KUKA KRL program: MyProgram_075().src

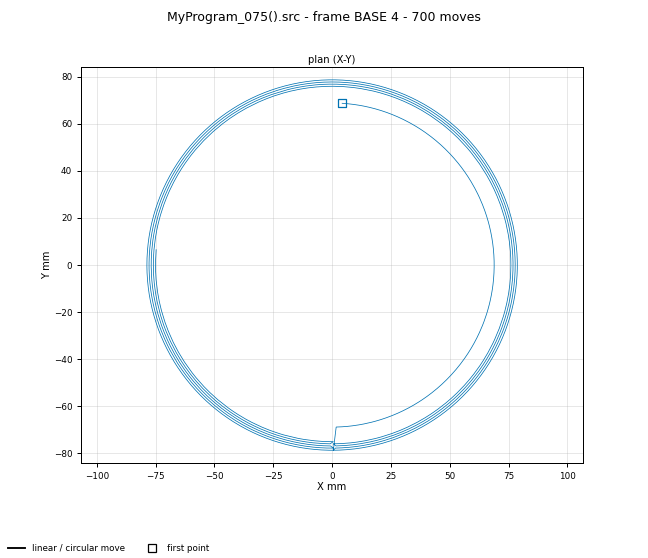
[picture p0: tool path of MyProgram_075().src in frame BASE 4, 700 of 700 moves have a stored position in this frame; points joined in program order, loops and branches not executed]
&ACCESS RVP
&REL 1
&PARAM TEMPLATE = C:\KRC\Roboter\Template\vorgabe
&PARAM EDITMASK = *
DEF MyProgram_075()
; ---- Setting reference (Base) ----
$BASE = BASE_DATA[4]

; --------------------------
; ---- Setting tool (TCP) ----
$TOOL = TOOL_DATA[3]
; --------------------------

$VEL.CP = VEL_APROX_PRINT
Startdeposition()
$VEL.CP = VEL_PRINT
LIN {X 4.2786,Y 68.757,Z 78,A 79.6597,B 24.8748,C -2.582,E1 25.012,E2 4.5437} C_DIS
LIN {X 6.8006,Y 68.5536,Z 78,A 77.5534,B 24.8748,C -2.5817,E1 25.0178,E2 6.6494} C_DIS
LIN {X 9.2868,Y 68.2614,Z 78,A 75.7343,B 24.8743,C -2.5876,E1 25.0228,E2 8.4531} C_DIS
LIN {X 11.7416,Y 67.8821,Z 78,A 73.6949,B 24.8743,C -2.5876,E1 25.0284,E2 10.4905} C_DIS
LIN {X 13.4915,Y 67.556,Z 78,A 72.2248,B 24.8743,C -2.5873,E1 25.0325,E2 11.9597} C_DIS
LIN {X 15.8736,Y 67.0363,Z 78,A 70.0908,B 24.8747,C -2.5836,E1 25.0383,E2 14.0995} C_DIS
LIN {X 18.4538,Y 66.3722,Z 78,A 67.9692,B 24.8746,C -2.5846,E1 25.044,E2 16.2154} C_DIS
LIN {X 20.828,Y 65.6662,Z 78,A 65.6223,B 24.8754,C -2.576,E1 25.0503,E2 18.5786} C_DIS
LIN {X 23.2331,Y 64.8543,Z 78,A 63.7895,B 24.8749,C -2.581,E1 25.0551,E2 20.3957} C_DIS
LIN {X 25.5953,Y 63.9589,Z 78,A 61.4087,B 24.8758,C -2.5721,E1 25.0614,E2 22.7926} C_DIS
LIN {X 27.9246,Y 62.9769,Z 78,A 59.3241,B 24.876,C -2.5702,E1 25.0667,E2 24.8765} C_DIS
LIN {X 30.2585,Y 61.8891,Z 78,A 57.1963,B 24.8762,C -2.568,E1 25.072,E2 27.0039} C_DIS
LIN {X 32.8695,Y 60.5417,Z 78,A 54.8407,B 24.8762,C -2.5671,E1 25.0779,E2 29.3552} C_DIS
LIN {X 35.4913,Y 59.0439,Z 78,A 52.275,B 24.8768,C -2.5621,E1 25.084,E2 31.9249} C_DIS
LIN {X 37.5793,Y 57.7379,Z 78,A 50.1926,B 24.8772,C -2.558,E1 25.0889,E2 34.0101} C_DIS
LIN {X 39.6743,Y 56.3189,Z 78,A 48.0936,B 24.8775,C -2.5547,E1 25.0938,E2 36.1097} C_DIS
LIN {X 42.0686,Y 54.5521,Z 78,A 45.8309,B 24.8774,C -2.5559,E1 25.0988,E2 38.3615} C_DIS
LIN {X 44.0446,Y 52.9696,Z 78,A 43.7356,B 24.8777,C -2.5522,E1 25.1033,E2 40.4575} C_DIS
LIN {X 46.2398,Y 51.0659,Z 78,A 41.2144,B 24.8784,C -2.5448,E1 25.1086,E2 42.9863} C_DIS
LIN {X 48.1387,Y 49.28,Z 78,A 38.9784,B 24.879,C -2.5386,E1 25.1131,E2 45.2277} C_DIS
LIN {X 50.2041,Y 47.1725,Z 78,A 36.7249,B 24.879,C -2.5386,E1 25.1175,E2 47.4716} C_DIS
LIN {X 51.888,Y 45.3137,Z 78,A 34.6568,B 24.8794,C -2.5344,E1 25.1213,E2 49.5403} C_DIS
LIN {X 53.5179,Y 43.3766,Z 78,A 32.5614,B 24.8799,C -2.5298,E1 25.125,E2 51.637} C_DIS
LIN {X 54.8494,Y 41.682,Z 78,A 30.5831,B 24.8807,C -2.5206,E1 25.1284,E2 53.6276} C_DIS
LIN {X 56.3431,Y 39.6397,Z 78,A 28.4879,B 24.8812,C -2.5156,E1 25.1318,E2 55.7244} C_DIS
LIN {X 57.7579,Y 37.5483,Z 78,A 26.6761,B 24.881,C -2.518,E1 25.1346,E2 57.5216} C_DIS
LIN {X 59.0958,Y 35.4055,Z 78,A 24.3033,B 24.8822,C -2.5053,E1 25.1381,E2 59.9124} C_DIS
LIN {X 60.625,Y 32.7158,Z 78,A 21.9754,B 24.8822,C -2.505,E1 25.1412,E2 62.2288} C_DIS
LIN {X 61.8865,Y 30.2638,Z 78,A 19.7787,B 24.8826,C -2.5013,E1 25.144,E2 64.4226} C_DIS
LIN {X 62.6469,Y 28.657,Z 78,A 18.0045,B 24.8837,C -2.4892,E1 25.1461,E2 66.2158} C_DIS
LIN {X 63.9379,Y 25.6469,Z 78,A 15.3278,B 24.8843,C -2.4827,E1 25.149,E2 68.8931} C_DIS
LIN {X 64.8826,Y 23.1535,Z 78,A 13.1121,B 24.8849,C -2.4763,E1 25.1511,E2 71.1115} C_DIS
LIN {X 65.6891,Y 20.7553,Z 78,A 11.0195,B 24.8855,C -2.4704,E1 25.1529,E2 73.2062} C_DIS
LIN {X 66.3949,Y 18.3737,Z 78,A 9.2251,B 24.8853,C -2.4716,E1 25.1543,E2 74.9876} C_DIS
LIN {X 66.836,Y 16.6972,Z 78,A 7.5223,B 24.8864,C -2.4601,E1 25.1555,E2 76.7076} C_DIS
LIN {X 67.3994,Y 14.2542,Z 78,A 5.7231,B 24.8863,C -2.4615,E1 25.1565,E2 78.493} C_DIS
LIN {X 67.869,Y 11.8169,Z 78,A 3.6106,B 24.887,C -2.4539,E1 25.1576,E2 80.6113} C_DIS
LIN {X 68.2635,Y 9.2719,Z 78,A 1.5451,B 24.8874,C -2.4493,E1 25.1585,E2 82.6754} C_DIS
LIN {X 68.5556,Y 6.7813,Z 78,A -0.5387,B 24.888,C -2.4428,E1 25.1591,E2 84.7622} C_DIS
LIN {X 68.7582,Y 4.2609,Z 78,A -2.6227,B 24.8886,C -2.4367,E1 25.1595,E2 86.8483} C_DIS
LIN {X 68.8683,Y 1.734,Z 78,A -4.7221,B 24.8892,C -2.4302,E1 25.1598,E2 88.9506} C_DIS
LIN {X 68.8856,Y -0.7727,Z 78,A -6.777,B 24.8897,C -2.4244,E1 25.1598,E2 91.007} C_DIS
LIN {X 68.8078,Y -3.3703,Z 78,A -8.9237,B 24.8903,C -2.4179,E1 25.1595,E2 93.1562} C_DIS
LIN {X 68.6402,Y -5.8623,Z 78,A -10.9954,B 24.8909,C -2.4114,E1 25.1591,E2 95.2308} C_DIS
LIN {X 68.3768,Y -8.3944,Z 78,A -13.0575,B 24.8913,C -2.4062,E1 25.1585,E2 97.2931} C_DIS
LIN {X 68.1372,Y -10.1567,Z 78,A -14.8223,B 24.8925,C -2.3937,E1 25.1578,E2 99.077} C_DIS
LIN {X 67.7274,Y -12.6047,Z 78,A -16.5998,B 24.8924,C -2.395,E1 25.1569,E2 100.841} C_DIS
LIN {X 67.2192,Y -15.0813,Z 78,A -18.6632,B 24.8929,C -2.3895,E1 25.1557,E2 102.9055} C_DIS
LIN {X 66.8248,Y -16.7427,Z 78,A -20.1027,B 24.8933,C -2.3845,E1 25.1548,E2 104.3485} C_DIS
LIN {X 66.1771,Y -19.1423,Z 78,A -22.1623,B 24.8939,C -2.3783,E1 25.1532,E2 106.411} C_DIS
LIN {X 65.6458,Y -20.8911,Z 78,A -23.9282,B 24.8949,C -2.3668,E1 25.1517,E2 108.1938} C_DIS
LIN {X 64.5825,Y -23.9782,Z 78,A -26.3411,B 24.8949,C -2.3668,E1 25.1495,E2 110.5934} C_DIS
LIN {X 63.9437,Y -25.6327,Z 78,A -28.0923,B 24.896,C -2.3548,E1 25.1477,E2 112.3632} C_DIS
LIN {X 62.6548,Y -28.6393,Z 78,A -30.5251,B 24.896,C -2.3545,E1 25.145,E2 114.7834} C_DIS
LIN {X 61.5438,Y -30.9551,Z 78,A -32.8114,B 24.8969,C -2.3441,E1 25.1421,E2 117.082} C_DIS
LIN {X 60.331,Y -33.2567,Z 78,A -34.7671,B 24.8969,C -2.3434,E1 25.1396,E2 119.029} C_DIS
LIN {X 59.111,Y -35.3799,Z 78,A -37.0001,B 24.8979,C -2.3323,E1 25.1364,E2 121.2768} C_DIS
LIN {X 57.7275,Y -37.5951,Z 78,A -39.257,B 24.8987,C -2.3239,E1 25.133,E2 123.5421} C_DIS
LIN {X 56.3166,Y -39.6775,Z 78,A -41.3446,B 24.8992,C -2.3183,E1 25.1297,E2 125.6327} C_DIS
LIN {X 54.5098,Y -42.1235,Z 78,A -43.8424,B 24.8997,C -2.3124,E1 25.1255,E2 128.1325} C_DIS
LIN {X 52.7111,Y -44.3556,Z 78,A -46.1758,B 24.9001,C -2.3076,E1 25.1213,E2 130.4666} C_DIS
LIN {X 50.7147,Y -46.6232,Z 78,A -48.7308,B 24.9007,C -2.3002,E1 25.1165,E2 133.0277} C_DIS
LIN {X 48.6926,Y -48.7328,Z 78,A -51.1426,B 24.9012,C -2.2948,E1 25.1118,E2 135.4421} C_DIS
LIN {X 46.5721,Y -50.7616,Z 78,A -53.3854,B 24.9012,C -2.2944,E1 25.1072,E2 137.6766} C_DIS
LIN {X 44.6488,Y -52.4613,Z 78,A -55.7017,B 24.9021,C -2.2847,E1 25.1023,E2 140.0066} C_DIS
LIN {X 42.3702,Y -54.3197,Z 78,A -57.8465,B 24.9018,C -2.2874,E1 25.0977,E2 142.1372} C_DIS
LIN {X 40.358,Y -55.831,Z 78,A -59.9287,B 24.9022,C -2.2833,E1 25.093,E2 144.2215} C_DIS
LIN {X 38.2711,Y -57.2817,Z 78,A -62.0044,B 24.9025,C -2.2801,E1 25.0882,E2 146.2977} C_DIS
LIN {X 36.8169,Y -58.2268,Z 78,A -63.7389,B 24.9034,C -2.2698,E1 25.0841,E2 148.0511} C_DIS
LIN {X 34.6799,Y -59.5246,Z 78,A -65.547,B 24.9031,C -2.273,E1 25.0798,E2 149.8459} C_DIS
LIN {X 32.4785,Y -60.7538,Z 78,A -67.8751,B 24.9039,C -2.2634,E1 25.0741,E2 152.1901} C_DIS
LIN {X 30.1975,Y -61.9191,Z 78,A -70.0366,B 24.9043,C -2.2592,E1 25.0686,E2 154.3557} C_DIS
LIN {X 27.9116,Y -62.9827,Z 78,A -71.8452,B 24.9039,C -2.2634,E1 25.0641,E2 156.1498} C_DIS
LIN {X 25.5875,Y -63.9621,Z 78,A -74.2251,B 24.9048,C -2.2532,E1 25.0579,E2 158.5485} C_DIS
LIN {X 23.1567,Y -64.8814,Z 78,A -76.352,B 24.9049,C -2.2512,E1 25.0523,E2 160.6755} C_DIS
LIN {X 20.757,Y -65.6885,Z 78,A -78.4536,B 24.9051,C -2.2488,E1 25.0467,E2 162.7789} C_DIS
LIN {X 18.3446,Y -66.4028,Z 78,A -80.2786,B 24.9047,C -2.2533,E1 25.0419,E2 164.5902} C_DIS
LIN {X 16.6718,Y -66.8422,Z 78,A -81.9846,B 24.9054,C -2.2451,E1 25.0372,E2 166.313} C_DIS
LIN {X 13.475,Y -67.5594,Z 78,A -84.4101,B 24.905,C -2.2502,E1 25.0306,E2 168.7233} C_DIS
LIN {X 11.3377,Y -67.9497,Z 78,A -86.3388,B 24.9054,C -2.2458,E1 25.0253,E2 170.6604} C_DIS
LIN {X 8.4843,Y -68.3656,Z 78,A -88.6117,B 24.9053,C -2.2473,E1 25.019,E2 172.9278} C_DIS
LIN {X 6.699,Y -68.5635,Z 78,A -90.3546,B 24.9058,C -2.2403,E1 25.0141,E2 174.6862} C_DIS
LIN {X 4.2094,Y -68.7615,Z 78,A -92.2011,B 24.9054,C -2.245,E1 25.009,E2 176.5206} C_DIS
LIN {X 1.7291,Y -68.8684,Z 78,A -94.2379,B 24.9054,C -2.245,E1 25.0033,E2 178.557} C_DIS
LIN {X 1.7291,Y -68.8684,Z 78,A -94.2379,B 24.9054,C -2.245,E1 25.0033,E2 178.557} C_DIS
Enddeposition()
LIN {X 0.524,Y -78.7317,Z 79,A -94.3644,B 24.917,C -2.1042,E1 25.002,E2 179.0178} C_DIS
Startdeposition()
$VEL.CP = VEL_PRINT
LIN {X -1.339,Y -78.7246,Z 79,A -96.4259,B 24.9186,C -2.0837,E1 24.9962,E2 181.1278} C_DIS
LIN {X -4.456,Y -78.6098,Z 79,A -98.6122,B 24.9184,C -2.0859,E1 24.9901,E2 183.3094} C_DIS
LIN {X -7.2304,Y -78.4032,Z 79,A -100.6782,B 24.9184,C -2.0848,E1 24.9843,E2 185.379} C_DIS
LIN {X -10.008,Y -78.0973,Z 79,A -102.7545,B 24.9186,C -2.0839,E1 24.9785,E2 187.4588} C_DIS
LIN {X -13.0934,Y -77.6397,Z 79,A -105.1259,B 24.9187,C -2.0817,E1 24.972,E2 189.8376} C_DIS
LIN {X -16.3074,Y -77.0302,Z 79,A -107.5052,B 24.9187,C -2.0826,E1 24.9655,E2 192.2173} C_DIS
LIN {X -19.4927,Y -76.2849,Z 79,A -109.7919,B 24.9184,C -2.0865,E1 24.9593,E2 194.498} C_DIS
LIN {X -22.4988,Y -75.453,Z 79,A -111.9817,B 24.9181,C -2.0902,E1 24.9534,E2 196.6825} C_DIS
LIN {X -25.2608,Y -74.5738,Z 79,A -114.0947,B 24.9179,C -2.0917,E1 24.9478,E2 198.7958} C_DIS
LIN {X -27.9886,Y -73.5935,Z 79,A -116.3922,B 24.9182,C -2.0885,E1 24.9418,E2 201.1057} C_DIS
LIN {X -31.0219,Y -72.3686,Z 79,A -118.7414,B 24.9179,C -2.0917,E1 24.9357,E2 203.4526} C_DIS
LIN {X -33.6646,Y -71.1778,Z 79,A -120.8891,B 24.9179,C -2.093,E1 24.9303,E2 205.6024} C_DIS
LIN {X -36.2616,Y -69.8904,Z 79,A -123.0044,B 24.9177,C -2.0955,E1 24.925,E2 207.7175} C_DIS
LIN {X -39.1328,Y -68.3226,Z 79,A -125.2953,B 24.9172,C -2.1011,E1 24.9194,E2 210.0017} C_DIS
LIN {X -41.8081,Y -66.7191,Z 79,A -127.4889,B 24.9168,C -2.1065,E1 24.9142,E2 212.1894} C_DIS
LIN {X -44.2355,Y -65.135,Z 79,A -129.7901,B 24.9169,C -2.1047,E1 24.9088,E2 214.5023} C_DIS
LIN {X -46.9038,Y -63.2425,Z 79,A -132.1761,B 24.9166,C -2.1086,E1 24.9034,E2 216.8875} C_DIS
LIN {X -49.1998,Y -61.4732,Z 79,A -134.2939,B 24.9163,C -2.1121,E1 24.8988,E2 219.0047} C_DIS
LIN {X -51.4291,Y -59.6206,Z 79,A -136.4121,B 24.916,C -2.1159,E1 24.8943,E2 221.1222} C_DIS
LIN {X -53.5887,Y -57.6873,Z 79,A -138.5308,B 24.9157,C -2.1198,E1 24.8899,E2 223.2401} C_DIS
LIN {X -55.9377,Y -55.4105,Z 79,A -140.8254,B 24.9152,C -2.127,E1 24.8854,E2 225.5272} C_DIS
LIN {X -58.0885,Y -53.1515,Z 79,A -143.0217,B 24.9146,C -2.1338,E1 24.8812,E2 227.7169} C_DIS
LIN {X -60.0055,Y -50.9774,Z 79,A -145.3272,B 24.9146,C -2.1335,E1 24.877,E2 230.0334} C_DIS
LIN {X -61.9167,Y -48.6387,Z 79,A -147.5039,B 24.9142,C -2.1392,E1 24.8732,E2 232.2067} C_DIS
LIN {X -63.8133,Y -46.1242,Z 79,A -149.8376,B 24.9138,C -2.1437,E1 24.8693,E2 234.5411} C_DIS
LIN {X -65.673,Y -43.4329,Z 79,A -152.1344,B 24.9132,C -2.1518,E1 24.8657,E2 236.8298} C_DIS
LIN {X -67.2271,Y -40.9862,Z 79,A -154.2559,B 24.9127,C -2.1569,E1 24.8626,E2 238.95} C_DIS
LIN {X -68.7977,Y -38.2914,Z 79,A -156.6403,B 24.9125,C -2.1601,E1 24.8593,E2 241.3393} C_DIS
LIN {X -70.3301,Y -35.4012,Z 79,A -158.9641,B 24.9118,C -2.168,E1 24.8563,E2 243.6568} C_DIS
LIN {X -71.5855,Y -32.7886,Z 79,A -161.1545,B 24.9115,C -2.1718,E1 24.8537,E2 245.8499} C_DIS
LIN {X -72.7439,Y -30.1315,Z 79,A -163.2772,B 24.9111,C -2.1775,E1 24.8514,E2 247.9708} C_DIS
LIN {X -73.8036,Y -27.4336,Z 79,A -165.4003,B 24.9106,C -2.1832,E1 24.8493,E2 250.0921} C_DIS
LIN {X -74.7634,Y -24.6985,Z 79,A -167.5235,B 24.9101,C -2.1891,E1 24.8474,E2 252.2134} C_DIS
LIN {X -75.7234,Y -21.5712,Z 79,A -169.8226,B 24.9094,C -2.1982,E1 24.8456,E2 254.5039} C_DIS
LIN {X -76.5184,Y -18.5551,Z 79,A -172.209,B 24.909,C -2.2022,E1 24.8439,E2 256.8948} C_DIS
LIN {X -77.2245,Y -15.3609,Z 79,A -174.6022,B 24.9085,C -2.2092,E1 24.8426,E2 259.2855} C_DIS
LIN {X -77.7375,Y -12.5081,Z 79,A -176.7265,B 24.9079,C -2.2154,E1 24.8416,E2 261.4077} C_DIS
LIN {X -78.1452,Y -9.6383,Z 79,A -178.8507,B 24.9074,C -2.2216,E1 24.8408,E2 263.5297} C_DIS
LIN {X -78.4768,Y -6.3838,Z 79,A 178.8495,B 24.9066,C -2.2311,E1 24.8402,E2 265.8206} C_DIS
LIN {X -78.668,Y -3.2706,Z 79,A 176.6473,B 24.9059,C -2.2399,E1 24.8399,E2 268.015} C_DIS
LIN {X -78.7351,Y -0.3728,Z 79,A 174.3378,B 24.9057,C -2.2417,E1 24.8398,E2 270.3341} C_DIS
LIN {X -78.684,Y 2.8981,Z 79,A 171.944,B 24.9051,C -2.2489,E1 24.84,E2 272.7252} C_DIS
LIN {X -78.4943,Y 6.1639,Z 79,A 169.6436,B 24.9043,C -2.2585,E1 24.8404,E2 275.0165} C_DIS
LIN {X -78.1886,Y 9.268,Z 79,A 167.4412,B 24.9036,C -2.2673,E1 24.841,E2 277.2109} C_DIS
LIN {X -77.8282,Y 11.9216,Z 79,A 165.395,B 24.9032,C -2.2711,E1 24.8419,E2 279.2603} C_DIS
LIN {X -77.295,Y 14.9948,Z 79,A 163.1928,B 24.9025,C -2.28,E1 24.8429,E2 281.4544} C_DIS
LIN {X -76.6907,Y 17.8297,Z 79,A 160.8836,B 24.9023,C -2.2817,E1 24.8444,E2 283.7731} C_DIS
LIN {X -75.8852,Y 21.0003,Z 79,A 158.4898,B 24.9017,C -2.2888,E1 24.8461,E2 286.1639} C_DIS
LIN {X -75.0608,Y 23.7792,Z 79,A 156.3656,B 24.9012,C -2.295,E1 24.8478,E2 288.2855} C_DIS
LIN {X -74.1347,Y 26.5258,Z 79,A 154.242,B 24.9007,C -2.3011,E1 24.8498,E2 290.4066} C_DIS
LIN {X -72.9676,Y 29.5818,Z 79,A 151.9425,B 24.8999,C -2.3103,E1 24.8521,E2 292.697} C_DIS
LIN {X -71.7539,Y 32.415,Z 79,A 149.5721,B 24.8995,C -2.3139,E1 24.8548,E2 295.0719} C_DIS
LIN {X -70.3301,Y 35.4012,Z 79,A 147.2313,B 24.8988,C -2.3226,E1 24.8576,E2 297.4045} C_DIS
LIN {X -68.9795,Y 37.9659,Z 79,A 145.1083,B 24.8983,C -2.3283,E1 24.8604,E2 299.5251} C_DIS
LIN {X -67.5353,Y 40.4791,Z 79,A 142.9176,B 24.8979,C -2.3323,E1 24.8635,E2 301.7176} C_DIS
LIN {X -65.7944,Y 43.2487,Z 79,A 140.6195,B 24.8972,C -2.341,E1 24.867,E2 304.0066} C_DIS
LIN {X -64.0298,Y 45.8207,Z 79,A 138.2347,B 24.8969,C -2.3443,E1 24.8708,E2 306.3952} C_DIS
LIN {X -62.0723,Y 48.4417,Z 79,A 135.9114,B 24.8962,C -2.352,E1 24.8747,E2 308.7112} C_DIS
LIN {X -60.2473,Y 50.6936,Z 79,A 133.722,B 24.8959,C -2.3554,E1 24.8786,E2 310.9025} C_DIS
LIN {X -58.3406,Y 52.8768,Z 79,A 131.601,B 24.8955,C -2.3604,E1 24.8826,E2 313.0211} C_DIS
LIN {X -56.0928,Y 55.2535,Z 79,A 129.3047,B 24.8947,C -2.3683,E1 24.887,E2 315.3085} C_DIS
LIN {X -53.8603,Y 57.4319,Z 79,A 127.1065,B 24.8941,C -2.3755,E1 24.8914,E2 317.4988} C_DIS
LIN {X -51.7099,Y 59.3754,Z 79,A 124.9864,B 24.8937,C -2.3799,E1 24.8958,E2 319.6166} C_DIS
LIN {X -49.6608,Y 61.0996,Z 79,A 122.9445,B 24.8935,C -2.3818,E1 24.9002,E2 321.6618} C_DIS
LIN {X -47.3783,Y 62.886,Z 79,A 120.8252,B 24.8932,C -2.386,E1 24.9049,E2 323.7789} C_DIS
LIN {X -44.8504,Y 64.7132,Z 79,A 118.4443,B 24.893,C -2.3877,E1 24.9104,E2 326.164} C_DIS
LIN {X -42.1243,Y 66.5216,Z 79,A 116.0571,B 24.8926,C -2.392,E1 24.9159,E2 328.5487} C_DIS
LIN {X -39.6473,Y 68.027,Z 79,A 113.9774,B 24.8922,C -2.3965,E1 24.9209,E2 330.6239} C_DIS
LIN {X -37.1165,Y 69.4402,Z 79,A 111.8299,B 24.892,C -2.3991,E1 24.9262,E2 332.7714} C_DIS
LIN {X -34.1995,Y 70.9207,Z 79,A 109.5301,B 24.8915,C -2.405,E1 24.9319,E2 335.0632} C_DIS
LIN {X -31.3636,Y 72.2196,Z 79,A 107.3364,B 24.891,C -2.4103,E1 24.9375,E2 337.2495} C_DIS
LIN {X -28.6842,Y 73.3251,Z 79,A 105.2206,B 24.8907,C -2.4131,E1 24.943,E2 339.3635} C_DIS
LIN {X -25.9659,Y 74.3312,Z 79,A 103.105,B 24.8905,C -2.4156,E1 24.9485,E2 341.4774} C_DIS
LIN {X -23.2123,Y 75.2366,Z 79,A 100.806,B 24.8907,C -2.413,E1 24.9547,E2 343.7866} C_DIS
LIN {X -20.0675,Y 76.1372,Z 79,A 98.4236,B 24.8905,C -2.4153,E1 24.9611,E2 346.1671} C_DIS
LIN {X -16.8872,Y 76.9037,Z 79,A 96.1349,B 24.8901,C -2.42,E1 24.9673,E2 348.4478} C_DIS
LIN {X -13.828,Y 77.5122,Z 79,A 93.9446,B 24.8897,C -2.4239,E1 24.9733,E2 350.6312} C_DIS
LIN {X -10.9656,Y 77.9686,Z 79,A 91.6483,B 24.8901,C -2.4203,E1 24.9796,E2 352.938} C_DIS
LIN {X -7.7176,Y 78.3582,Z 79,A 89.2683,B 24.89,C -2.4215,E1 24.9862,E2 355.3165} C_DIS
LIN {X -4.456,Y 78.6098,Z 79,A 86.9822,B 24.8896,C -2.4251,E1 24.9926,E2 357.5949} C_DIS
LIN {X -1.339,Y 78.7246,Z 79,A 84.7943,B 24.8894,C -2.428,E1 24.9987,E2 359.7762} C_DIS
LIN {X 1.339,Y 78.7246,Z 79,A 82.7613,B 24.8895,C -2.426,E1 25.0044,E2 361.8138} C_DIS
LIN {X 4.456,Y 78.6098,Z 79,A 80.5744,B 24.8893,C -2.4284,E1 25.0104,E2 363.9943} C_DIS
LIN {X 7.3464,Y 78.3925,Z 79,A 78.4655,B 24.8893,C -2.4283,E1 25.0163,E2 366.1024} C_DIS
LIN {X 10.008,Y 78.0973,Z 79,A 76.434,B 24.8896,C -2.4256,E1 25.022,E2 368.1387} C_DIS
LIN {X 13.0562,Y 77.6459,Z 79,A 74.0814,B 24.8899,C -2.4218,E1 25.0285,E2 370.498} C_DIS
LIN {X 16.3074,Y 77.0302,Z 79,A 71.6907,B 24.8899,C -2.4213,E1 25.035,E2 372.8871} C_DIS
LIN {X 19.4927,Y 76.2849,Z 79,A 69.4096,B 24.8899,C -2.4228,E1 25.0412,E2 375.1613} C_DIS
LIN {X 22.4988,Y 75.453,Z 79,A 67.0431,B 24.8902,C -2.4184,E1 25.0475,E2 377.5341} C_DIS
LIN {X 25.6141,Y 74.4547,Z 79,A 64.6703,B 24.8904,C -2.4167,E1 25.0538,E2 379.9065} C_DIS
LIN {X 28.3372,Y 73.4614,Z 79,A 62.6491,B 24.8904,C -2.4172,E1 25.0591,E2 381.922} C_DIS
LIN {X 31.0219,Y 72.3686,Z 79,A 60.4608,B 24.8908,C -2.4128,E1 25.0648,E2 384.1158} C_DIS
LIN {X 33.6542,Y 71.1826,Z 79,A 58.3643,B 24.891,C -2.4105,E1 25.0701,E2 386.2125} C_DIS
LIN {X 36.2616,Y 69.8904,Z 79,A 56.2534,B 24.8912,C -2.408,E1 25.0753,E2 388.3235} C_DIS
LIN {X 39.1328,Y 68.3226,Z 79,A 53.9766,B 24.8912,C -2.4077,E1 25.0809,E2 390.5942} C_DIS
LIN {X 41.8081,Y 66.7191,Z 79,A 51.7974,B 24.8912,C -2.407,E1 25.086,E2 392.7682} C_DIS
LIN {X 44.2355,Y 65.135,Z 79,A 49.6953,B 24.8916,C -2.4039,E1 25.0909,E2 394.8708} C_DIS
LIN {X 46.603,Y 63.4627,Z 79,A 47.5939,B 24.8919,C -2.4005,E1 25.0957,E2 396.9728} C_DIS
LIN {X 48.9073,Y 61.7044,Z 79,A 45.4929,B 24.8922,C -2.397,E1 25.1003,E2 399.0744} C_DIS
LIN {X 51.1453,Y 59.8624,Z 79,A 43.3923,B 24.8925,C -2.3933,E1 25.1048,E2 401.1757} C_DIS
LIN {X 53.3141,Y 57.9393,Z 79,A 41.2922,B 24.8929,C -2.3894,E1 25.1092,E2 403.2766} C_DIS
LIN {X 55.2535,Y 56.0928,Z 79,A 39.2694,B 24.8934,C -2.3832,E1 25.1133,E2 405.3057} C_DIS
LIN {X 57.4319,Y 53.8603,Z 79,A 37.0931,B 24.8936,C -2.3811,E1 25.1175,E2 407.4775} C_DIS
LIN {X 59.2303,Y 51.8761,Z 79,A 35.0713,B 24.8942,C -2.3745,E1 25.1213,E2 409.5059} C_DIS
LIN {X 61.2385,Y 49.4894,Z 79,A 32.8958,B 24.8944,C -2.3721,E1 25.1251,E2 411.6771} C_DIS
LIN {X 63.0186,Y 47.2019,Z 79,A 30.6151,B 24.8953,C -2.3618,E1 25.129,E2 413.9712} C_DIS
LIN {X 64.926,Y 44.5442,Z 79,A 28.2512,B 24.8958,C -2.3564,E1 25.1328,E2 416.3364} C_DIS
LIN {X 66.7191,Y 41.8081,Z 79,A 25.9802,B 24.8961,C -2.3536,E1 25.1362,E2 418.6025} C_DIS
LIN {X 68.2127,Y 39.3241,Z 79,A 23.883,B 24.8965,C -2.3484,E1 25.1392,E2 420.7012} C_DIS
LIN {X 69.6139,Y 36.7867,Z 79,A 21.7864,B 24.897,C -2.3431,E1 25.142,E2 422.7993} C_DIS
LIN {X 71.0163,Y 34.0006,Z 79,A 19.613,B 24.8973,C -2.3398,E1 25.1447,E2 424.969} C_DIS
LIN {X 72.0905,Y 31.66,Z 79,A 17.6233,B 24.8981,C -2.331,E1 25.147,E2 426.9687} C_DIS
LIN {X 73.3251,Y 28.6842,Z 79,A 15.2386,B 24.8987,C -2.323,E1 25.1495,E2 429.3591} C_DIS
LIN {X 74.4547,Y 25.6141,Z 79,A 12.8769,B 24.8993,C -2.3166,E1 25.1517,E2 431.7227} C_DIS
LIN {X 75.347,Y 22.8563,Z 79,A 10.7814,B 24.8998,C -2.3107,E1 25.1534,E2 433.8201} C_DIS
LIN {X 76.1372,Y 20.0675,Z 79,A 8.6862,B 24.9003,C -2.3048,E1 25.1549,E2 435.9173} C_DIS
LIN {X 76.9037,Y 16.8872,Z 79,A 6.42,B 24.9007,C -2.3011,E1 25.1564,E2 438.179} C_DIS
LIN {X 77.5122,Y 13.828,Z 79,A 4.2458,B 24.901,C -2.2971,E1 25.1575,E2 440.3501} C_DIS
LIN {X 77.9686,Y 10.9656,Z 79,A 1.9689,B 24.902,C -2.2853,E1 25.1585,E2 442.6414} C_DIS
LIN {X 78.3582,Y 7.7176,Z 79,A -0.391,B 24.9026,C -2.2784,E1 25.1592,E2 445.0036} C_DIS
LIN {X 78.5892,Y 4.8282,Z 79,A -2.4865,B 24.9031,C -2.2722,E1 25.1596,E2 447.1013} C_DIS
LIN {X 78.7137,Y 1.9323,Z 79,A -4.5809,B 24.9037,C -2.266,E1 25.1598,E2 449.1979} C_DIS
LIN {X 78.7246,Y -1.339,Z 79,A -6.7707,B 24.9038,C -2.2644,E1 25.1598,E2 451.3785} C_DIS
LIN {X 78.6257,Y -4.1677,Z 79,A -8.9234,B 24.9046,C -2.2549,E1 25.1595,E2 453.5408} C_DIS
LIN {X 78.4055,Y -7.2052,Z 79,A -11.0277,B 24.9049,C -2.2513,E1 25.159,E2 455.6411} C_DIS
LIN {X 78.0973,Y -10.008,Z 79,A -13.1325,B 24.9056,C -2.2431,E1 25.1583,E2 457.7528} C_DIS
LIN {X 77.6397,Y -13.0934,Z 79,A -15.4859,B 24.9064,C -2.2333,E1 25.1573,E2 460.1155} C_DIS
LIN {X 77.0302,Y -16.3074,Z 79,A -17.8464,B 24.907,C -2.2264,E1 25.156,E2 462.4786} C_DIS
LIN {X 76.2849,Y -19.4927,Z 79,A -20.1145,B 24.9073,C -2.2224,E1 25.1545,E2 464.7429} C_DIS
LIN {X 75.453,Y -22.4988,Z 79,A -22.286,B 24.9077,C -2.2184,E1 25.1528,E2 466.9115} C_DIS
LIN {X 74.5738,Y -25.2608,Z 79,A -24.381,B 24.9082,C -2.2123,E1 25.151,E2 469.009} C_DIS
LIN {X 73.5935,Y -27.9886,Z 79,A -26.6584,B 24.9092,C -2.2006,E1 25.1488,E2 471.3013} C_DIS
LIN {X 72.3686,Y -31.0219,Z 79,A -29.0195,B 24.9097,C -2.194,E1 25.1462,E2 473.6651} C_DIS
LIN {X 71.1778,Y -33.6646,Z 79,A -31.1148,B 24.9102,C -2.1881,E1 25.1438,E2 475.7628} C_DIS
LIN {X 69.8904,Y -36.2616,Z 79,A -33.2105,B 24.9107,C -2.1823,E1 25.1411,E2 477.8611} C_DIS
LIN {X 68.3226,Y -39.1328,Z 79,A -35.48,B 24.9109,C -2.1789,E1 25.138,E2 480.1268} C_DIS
LIN {X 66.7191,Y -41.8081,Z 79,A -37.6528,B 24.9112,C -2.1755,E1 25.1349,E2 482.2966} C_DIS
LIN {X 65.135,Y -44.2355,Z 79,A -39.9317,B 24.9121,C -2.1644,E1 25.1313,E2 484.5905} C_DIS
LIN {X 63.2425,Y -46.9038,Z 79,A -42.2946,B 24.9126,C -2.1585,E1 25.1275,E2 486.9559} C_DIS
LIN {X 61.5192,Y -49.1416,Z 79,A -44.3472,B 24.913,C -2.1531,E1 25.1239,E2 489.0115} C_DIS
LIN {X 59.6206,Y -51.4291,Z 79,A -46.4889,B 24.9134,C -2.1482,E1 25.12,E2 491.1551} C_DIS
LIN {X 57.6873,Y -53.5887,Z 79,A -48.5866,B 24.9138,C -2.1433,E1 25.1161,E2 493.2551} C_DIS
LIN {X 55.4105,Y -55.9377,Z 79,A -50.8584,B 24.914,C -2.1409,E1 25.1116,E2 495.5229} C_DIS
LIN {X 53.1515,Y -58.0885,Z 79,A -53.0338,B 24.9142,C -2.1384,E1 25.1072,E2 497.6952} C_DIS
LIN {X 50.9774,Y -60.0055,Z 79,A -55.3151,B 24.915,C -2.1284,E1 25.1024,E2 499.9912} C_DIS
LIN {X 48.4417,Y -62.0723,Z 79,A -57.6138,B 24.9153,C -2.1257,E1 25.0974,E2 502.2877} C_DIS
LIN {X 46.1242,Y -63.8133,Z 79,A -59.7805,B 24.9157,C -2.1196,E1 25.0925,E2 504.4611} C_DIS
LIN {X 43.4329,Y -65.673,Z 79,A -62.0545,B 24.9159,C -2.1182,E1 25.0872,E2 506.7309} C_DIS
LIN {X 40.9862,Y -67.2271,Z 79,A -64.1551,B 24.9161,C -2.1145,E1 25.0822,E2 508.8336} C_DIS
LIN {X 38.2914,Y -68.7977,Z 79,A -66.516,B 24.9167,C -2.1077,E1 25.0765,E2 511.2034} C_DIS
LIN {X 35.4012,Y -70.3301,Z 79,A -68.794,B 24.9167,C -2.1068,E1 25.0708,E2 513.4773} C_DIS
LIN {X 32.7886,Y -71.5855,Z 79,A -70.9865,B 24.9172,C -2.101,E1 25.0653,E2 515.6778} C_DIS
LIN {X 30.1315,Y -72.7439,Z 79,A -73.0889,B 24.9174,C -2.0982,E1 25.0599,E2 517.782} C_DIS
LIN {X 27.4336,Y -73.8036,Z 79,A -75.192,B 24.9177,C -2.0955,E1 25.0544,E2 519.8869} C_DIS
LIN {X 24.6985,Y -74.7634,Z 79,A -77.2955,B 24.9178,C -2.093,E1 25.0488,E2 521.992} C_DIS
LIN {X 21.5712,Y -75.7234,Z 79,A -79.5736,B 24.9178,C -2.0934,E1 25.0427,E2 524.2655} C_DIS
LIN {X 18.5551,Y -76.5184,Z 79,A -81.9386,B 24.9182,C -2.0883,E1 25.0363,E2 526.6389} C_DIS
LIN {X 15.3609,Y -77.2245,Z 79,A -84.3109,B 24.9184,C -2.0864,E1 25.0298,E2 529.0125} C_DIS
LIN {X 12.5081,Y -77.7375,Z 79,A -86.4169,B 24.9184,C -2.0849,E1 25.024,E2 531.12} C_DIS
LIN {X 9.6383,Y -78.1452,Z 79,A -88.5233,B 24.9186,C -2.0837,E1 25.0182,E2 533.2277} C_DIS
LIN {X 6.3838,Y -78.4768,Z 79,A -90.8044,B 24.9185,C -2.0853,E1 25.0118,E2 535.5036} C_DIS
LIN {X 3.2706,Y -78.668,Z 79,A -93.1719,B 24.9187,C -2.0816,E1 25.0052,E2 537.879} C_DIS
LIN {X 0.524,Y -78.7317,Z 79,A -94.3641,B 24.917,C -2.1041,E1 25.0021,E2 539.0176} C_DIS
Enddeposition()
LIN {X 0.524,Y -78.7317,Z 79,A -94.3641,B 24.917,C -2.1041,E1 25.0021,E2 539.0176} C_DIS
Startdeposition()
$VEL.CP = VEL_PRINT
LIN {X 1.4129,Y -77.8112,Z 79,A -93.6485,B 24.9156,C -2.1218,E1 25.0042,E2 538.2602} C_DIS
LIN {X 4.0715,Y -77.7178,Z 79,A -91.4974,B 24.9151,C -2.128,E1 25.0102,E2 536.095} C_DIS
LIN {X 7.2735,Y -77.4835,Z 79,A -89.0671,B 24.9148,C -2.1311,E1 25.017,E2 533.6587} C_DIS
LIN {X 10.6001,Y -77.0996,Z 79,A -86.6779,B 24.9148,C -2.1304,E1 25.0236,E2 531.2729} C_DIS
LIN {X 12.9926,Y -76.732,Z 79,A -84.8499,B 24.9147,C -2.1331,E1 25.0286,E2 529.4404} C_DIS
LIN {X 16.0464,Y -76.1528,Z 79,A -82.5167,B 24.9144,C -2.1363,E1 25.035,E2 527.1024} C_DIS
LIN {X 18.9409,Y -75.4852,Z 79,A -80.2864,B 24.9141,C -2.1397,E1 25.0411,E2 524.8673} C_DIS
LIN {X 22.1682,Y -74.6,Z 79,A -77.7363,B 24.9137,C -2.145,E1 25.048,E2 522.309} C_DIS
LIN {X 26.076,Y -73.3262,Z 79,A -74.4312,B 24.9127,C -2.1571,E1 25.0568,E2 518.9818} C_DIS
LIN {X 31.9189,Y -70.9772,Z 79,A -70.6081,B 24.9142,C -2.1395,E1 25.0665,E2 515.2093} C_DIS
LIN {X 35.1195,Y -69.4501,Z 79,A -67.6373,B 24.9129,C -2.1544,E1 25.074,E2 512.2111} C_DIS
LIN {X 38.1815,Y -67.8147,Z 79,A -65.2304,B 24.9129,C -2.1544,E1 25.0799,E2 509.8113} C_DIS
LIN {X 40.7785,Y -66.2863,Z 79,A -62.9274,B 24.9124,C -2.1609,E1 25.0854,E2 507.4998} C_DIS
LIN {X 43.2873,Y -64.6759,Z 79,A -60.678,B 24.9119,C -2.1668,E1 25.0907,E2 505.2439} C_DIS
LIN {X 45.711,Y -62.9857,Z 79,A -58.5678,B 24.9117,C -2.1693,E1 25.0955,E2 503.1352} C_DIS
LIN {X 48.3224,Y -61.0044,Z 79,A -56.179,B 24.9114,C -2.1737,E1 25.1007,E2 500.7448} C_DIS
LIN {X 50.8111,Y -58.9493,Z 79,A -53.7704,B 24.9109,C -2.18,E1 25.1059,E2 498.3307} C_DIS
LIN {X 53.2125,Y -56.7893,Z 79,A -51.5383,B 24.9108,C -2.181,E1 25.1105,E2 496.1051} C_DIS
LIN {X 55.4014,Y -54.6559,Z 79,A -49.303,B 24.9104,C -2.186,E1 25.1149,E2 493.8675} C_DIS
LIN {X 57.6319,Y -52.3003,Z 79,A -46.7958,B 24.9096,C -2.1956,E1 25.1197,E2 491.3487} C_DIS
LIN {X 59.627,Y -50.0133,Z 79,A -44.5986,B 24.9092,C -2.2002,E1 25.1237,E2 489.1506} C_DIS
LIN {X 61.2285,Y -48.0388,Z 79,A -42.6937,B 24.9087,C -2.2061,E1 25.127,E2 487.2405} C_DIS
LIN {X 63.1847,Y -45.4352,Z 79,A -40.3966,B 24.9084,C -2.2095,E1 25.1308,E2 484.9466} C_DIS
LIN {X 64.88,Y -42.9789,Z 79,A -38.248,B 24.908,C -2.214,E1 25.1341,E2 482.7979} C_DIS
LIN {X 66.2261,Y -40.8761,Z 79,A -36.3083,B 24.9074,C -2.2224,E1 25.137,E2 480.8483} C_DIS
LIN {X 67.8422,Y -38.1322,Z 79,A -34.105,B 24.9072,C -2.2247,E1 25.1401,E2 478.6508} C_DIS
LIN {X 69.4059,Y -35.2059,Z 79,A -31.3104,B 24.9056,C -2.2429,E1 25.1437,E2 475.8281} C_DIS
LIN {X 70.6903,Y -32.5509,Z 79,A -28.9185,B 24.9045,C -2.2563,E1 25.1465,E2 473.4175} C_DIS
LIN {X 72.4833,Y -28.3331,Z 79,A -26.1825,B 24.9053,C -2.2464,E1 25.1494,E2 470.7199} C_DIS
LIN {X 73.2368,Y -26.3264,Z 79,A -24.371,B 24.9043,C -2.2586,E1 25.1511,E2 468.8898} C_DIS
LIN {X 74.4776,Y -22.5807,Z 79,A -21.5751,B 24.9038,C -2.2641,E1 25.1535,E2 466.0967} C_DIS
LIN {X 75.3226,Y -19.5737,Z 79,A -19.4145,B 24.9036,C -2.267,E1 25.155,E2 463.9417} C_DIS
LIN {X 75.9066,Y -17.1726,Z 79,A -17.6712,B 24.9033,C -2.2703,E1 25.1561,E2 462.2007} C_DIS
LIN {X 76.4961,Y -14.321,Z 79,A -15.3847,B 24.9023,C -2.2816,E1 25.1574,E2 459.901} C_DIS
LIN {X 77.1956,Y -9.8707,Z 79,A -11.8227,B 24.9008,C -2.2999,E1 25.1588,E2 456.3167} C_DIS
LIN {X 77.6193,Y -5.6559,Z 79,A -9.01,B 24.9008,C -2.3002,E1 25.1595,E2 453.52} C_DIS
LIN {X 77.7777,Y -2.7033,Z 79,A -6.8582,B 24.9002,C -2.3063,E1 25.1597,E2 451.3665} C_DIS
LIN {X 77.8231,Y 0.3922,Z 79,A -4.7156,B 24.8999,C -2.3093,E1 25.1597,E2 449.2296} C_DIS
LIN {X 77.7517,Y 3.355,Z 79,A -2.4303,B 24.8991,C -2.3195,E1 25.1596,E2 446.9339} C_DIS
LIN {X 77.5499,Y 6.5345,Z 79,A -0.1123,B 24.8985,C -2.326,E1 25.1591,E2 444.6142} C_DIS
LIN {X 77.2199,Y 9.6834,Z 79,A 2.2191,B 24.8978,C -2.3333,E1 25.1583,E2 442.2793} C_DIS
LIN {X 76.7379,Y 12.9574,Z 79,A 4.6553,B 24.8972,C -2.3409,E1 25.1573,E2 439.8395} C_DIS
LIN {X 76.0881,Y 16.3476,Z 79,A 7.2107,B 24.8965,C -2.3491,E1 25.1558,E2 437.2795} C_DIS
LIN {X 75.3446,Y 19.4882,Z 79,A 9.5101,B 24.896,C -2.354,E1 25.1543,E2 434.982} C_DIS
LIN {X 74.4783,Y 22.5776,Z 79,A 12.0168,B 24.895,C -2.3655,E1 25.1523,E2 432.4623} C_DIS
LIN {X 73.2947,Y 26.1656,Z 79,A 15.3837,B 24.8926,C -2.392,E1 25.1491,E2 429.0518} C_DIS
LIN {X 71.9416,Y 29.6812,Z 79,A 17.354,B 24.8942,C -2.3749,E1 25.1471,E2 427.1327} C_DIS
LIN {X 70.7618,Y 32.3965,Z 79,A 19.6007,B 24.8934,C -2.3831,E1 25.1446,E2 424.8789} C_DIS
LIN {X 69.4429,Y 35.1335,Z 79,A 21.7826,B 24.893,C -2.3876,E1 25.1419,E2 422.6981} C_DIS
LIN {X 68.023,Y 37.8084,Z 79,A 23.6309,B 24.8935,C -2.3819,E1 25.1394,E2 420.8729} C_DIS
LIN {X 66.6953,Y 40.1056,Z 79,A 25.9773,B 24.892,C -2.3991,E1 25.1361,E2 418.4979} C_DIS
LIN {X 64.9072,Y 42.9378,Z 79,A 28.4078,B 24.8915,C -2.4043,E1 25.1324,E2 416.0672} C_DIS
LIN {X 63.0434,Y 45.6322,Z 79,A 30.9193,B 24.8907,C -2.4133,E1 25.1283,E2 413.5467} C_DIS
LIN {X 60.8826,Y 48.4764,Z 79,A 33.4624,B 24.8904,C -2.417,E1 25.1239,E2 411.007} C_DIS
LIN {X 58.7445,Y 51.0461,Z 79,A 35.8063,B 24.8902,C -2.4191,E1 25.1197,E2 408.6688} C_DIS
LIN {X 56.6041,Y 53.4095,Z 79,A 37.9935,B 24.8902,C -2.4194,E1 25.1156,E2 406.4904} C_DIS
LIN {X 54.5859,Y 55.4706,Z 79,A 40.306,B 24.8892,C -2.4295,E1 25.111,E2 404.1638} C_DIS
LIN {X 52.2212,Y 57.7036,Z 79,A 42.7046,B 24.8888,C -2.4345,E1 25.1061,E2 401.7632} C_DIS
LIN {X 49.8166,Y 59.7905,Z 79,A 44.9641,B 24.8886,C -2.4364,E1 25.1013,E2 399.5078} C_DIS
LIN {X 47.357,Y 61.757,Z 79,A 47.057,B 24.8888,C -2.4339,E1 25.0967,E2 397.4287} C_DIS
LIN {X 44.8502,Y 63.6021,Z 79,A 49.6599,B 24.8876,C -2.447,E1 25.0908,E2 394.8039} C_DIS
LIN {X 42.2301,Y 65.3701,Z 79,A 51.9041,B 24.8876,C -2.4483,E1 25.0856,E2 392.5642} C_DIS
LIN {X 39.3149,Y 67.1642,Z 79,A 54.4837,B 24.887,C -2.4537,E1 25.0794,E2 389.9797} C_DIS
LIN {X 35.9329,Y 69.033,Z 79,A 57.3198,B 24.8867,C -2.4572,E1 25.0724,E2 387.1434} C_DIS
LIN {X 32.6565,Y 70.6412,Z 79,A 59.9843,B 24.8864,C -2.4598,E1 25.0657,E2 384.4798} C_DIS
LIN {X 29.8877,Y 71.8571,Z 79,A 62.0146,B 24.8867,C -2.4565,E1 25.0605,E2 382.4622} C_DIS
LIN {X 27.063,Y 72.9682,Z 79,A 64.4435,B 24.886,C -2.4642,E1 25.0541,E2 380.0202} C_DIS
LIN {X 23.9794,Y 74.0376,Z 79,A 66.6874,B 24.8863,C -2.4616,E1 25.0482,E2 377.7867} C_DIS
LIN {X 21.1369,Y 74.8987,Z 79,A 68.9618,B 24.8859,C -2.4657,E1 25.0421,E2 375.5066} C_DIS
LIN {X 18.104,Y 75.6898,Z 79,A 71.3063,B 24.8857,C -2.468,E1 25.0358,E2 373.16} C_DIS
LIN {X 15.0244,Y 76.3606,Z 79,A 73.6164,B 24.8857,C -2.4688,E1 25.0294,E2 370.851} C_DIS
LIN {X 11.7894,Y 76.9259,Z 79,A 76.0268,B 24.8855,C -2.4694,E1 25.0228,E2 368.4416} C_DIS
LIN {X 8.5804,Y 77.351,Z 79,A 78.4828,B 24.8853,C -2.4718,E1 25.016,E2 365.9817} C_DIS
LIN {X 5.8675,Y 77.6033,Z 79,A 80.3409,B 24.8857,C -2.4679,E1 25.0108,E2 364.134} C_DIS
LIN {X 2.9078,Y 77.7708,Z 79,A 82.6288,B 24.8854,C -2.4707,E1 25.0044,E2 361.8401} C_DIS
LIN {X -0.2748,Y 77.8238,Z 79,A 84.9027,B 24.8856,C -2.4684,E1 24.9981,E2 359.5719} C_DIS
LIN {X -3.4315,Y 77.7484,Z 79,A 87.1117,B 24.886,C -2.4645,E1 24.992,E2 357.3718} C_DIS
LIN {X -6.4015,Y 77.5606,Z 79,A 89.5998,B 24.8853,C -2.4717,E1 24.985,E2 354.8655} C_DIS
LIN {X -10.01,Y 77.1776,Z 79,A 92.0242,B 24.8861,C -2.4634,E1 24.9783,E2 352.4591} C_DIS
LIN {X -13.1857,Y 76.6997,Z 79,A 94.4818,B 24.8861,C -2.4643,E1 24.9715,E2 349.9972} C_DIS
LIN {X -16.0978,Y 76.1412,Z 79,A 97.0951,B 24.8851,C -2.4741,E1 24.9643,E2 347.3574} C_DIS
LIN {X -20.3081,Y 75.1276,Z 79,A 99.8083,B 24.8866,C -2.4583,E1 24.9571,E2 344.6782} C_DIS
LIN {X -23.4427,Y 74.2105,Z 79,A 102.0296,B 24.8873,C -2.4507,E1 24.9512,E2 342.471} C_DIS
LIN {X -27.7006,Y 72.7274,Z 79,A 105.6939,B 24.8868,C -2.4557,E1 24.9415,E2 338.7877} C_DIS
LIN {X -31.2436,Y 71.2772,Z 79,A 108.4693,B 24.8873,C -2.4505,E1 24.9343,E2 336.0182} C_DIS
LIN {X -34.0145,Y 69.998,Z 79,A 110.8154,B 24.8873,C -2.4497,E1 24.9284,E2 333.6682} C_DIS
LIN {X -36.1326,Y 68.9278,Z 79,A 113.2327,B 24.886,C -2.4644,E1 24.9224,E2 331.209} C_DIS
LIN {X -39.4755,Y 67.0693,Z 79,A 115.2469,B 24.8884,C -2.4384,E1 24.9176,E2 329.2507} C_DIS
LIN {X -42.1669,Y 65.4107,Z 79,A 117.6373,B 24.8887,C -2.4357,E1 24.912,E2 326.859} C_DIS
LIN {X -45.9431,Y 62.8157,Z 79,A 121.0617,B 24.8891,C -2.4304,E1 24.9042,E2 323.4358} C_DIS
LIN {X -48.6268,Y 60.7638,Z 79,A 123.5971,B 24.8895,C -2.4263,E1 24.8986,E2 320.9007} C_DIS
LIN {X -51.1932,Y 58.616,Z 79,A 125.939,B 24.8903,C -2.4178,E1 24.8936,E2 318.5701} C_DIS
LIN {X -53.1146,Y 56.8814,Z 79,A 127.9377,B 24.8905,C -2.4157,E1 24.8895,E2 316.5681} C_DIS
LIN {X -55.7977,Y 54.2523,Z 79,A 130.7454,B 24.891,C -2.4102,E1 24.884,E2 313.7618} C_DIS
LIN {X -58.0876,Y 51.7923,Z 79,A 133.1869,B 24.8916,C -2.4032,E1 24.8794,E2 311.326} C_DIS
LIN {X -60.1926,Y 49.3316,Z 79,A 135.8813,B 24.8915,C -2.4049,E1 24.8746,E2 308.6152} C_DIS
LIN {X -62.4757,Y 46.4057,Z 79,A 138.1942,B 24.8931,C -2.3871,E1 24.8707,E2 306.3337} C_DIS
LIN {X -64.2861,Y 43.8623,Z 79,A 140.8703,B 24.8928,C -2.3904,E1 24.8664,E2 303.6366} C_DIS
LIN {X -66.0463,Y 41.164,Z 79,A 143.7387,B 24.8922,C -2.3962,E1 24.8621,E2 300.7396} C_DIS
LIN {X -67.9119,Y 38.0073,Z 79,A 145.7177,B 24.8946,C -2.3704,E1 24.8595,E2 298.8119} C_DIS
LIN {X -69.5046,Y 35.0128,Z 79,A 148.4533,B 24.8946,C -2.3691,E1 24.856,E2 296.0649} C_DIS
LIN {X -71.0278,Y 31.8066,Z 79,A 150.7045,B 24.8962,C -2.3523,E1 24.8534,E2 293.8414} C_DIS
LIN {X -72.128,Y 29.2259,Z 79,A 152.7682,B 24.8967,C -2.3461,E1 24.8511,E2 291.7811} C_DIS
LIN {X -72.934,Y 27.1542,Z 79,A 154.8758,B 24.8961,C -2.3527,E1 24.849,E2 289.6458} C_DIS
LIN {X -74.431,Y 22.7298,Z 79,A 157.9027,B 24.898,C -2.332,E1 24.8465,E2 286.6512} C_DIS
LIN {X -75.1613,Y 20.1835,Z 79,A 160.0246,B 24.8981,C -2.3301,E1 24.8449,E2 284.5214} C_DIS
LIN {X -75.9421,Y 17.0168,Z 79,A 162.5203,B 24.8986,C -2.3249,E1 24.8433,E2 282.0235} C_DIS
LIN {X -76.573,Y 13.8986,Z 79,A 164.7275,B 24.8995,C -2.3142,E1 24.8421,E2 279.8289} C_DIS
LIN {X -77.0309,Y 11.0837,Z 79,A 166.8932,B 24.9,C -2.3092,E1 24.8412,E2 277.6623} C_DIS
LIN {X -77.4726,Y 7.3918,Z 79,A 169.6402,B 24.9007,C -2.3007,E1 24.8404,E2 274.9191} C_DIS
LIN {X -77.7235,Y 3.9689,Z 79,A 172.2324,B 24.9012,C -2.2942,E1 24.8399,E2 272.3267} C_DIS
LIN {X -77.8204,Y 0.8238,Z 79,A 174.5713,B 24.9018,C -2.2874,E1 24.8398,E2 269.99} C_DIS
LIN {X -77.8075,Y -1.6134,Z 79,A 176.267,B 24.9025,C -2.2793,E1 24.8398,E2 268.3034} C_DIS
LIN {X -77.6837,Y -4.6882,Z 79,A 178.6462,B 24.9029,C -2.2749,E1 24.8402,E2 265.9204} C_DIS
LIN {X -77.4365,Y -7.7647,Z 79,A -179.0332,B 24.9034,C -2.269,E1 24.8408,E2 263.6001} C_DIS
LIN {X -77.0605,Y -10.8746,Z 79,A -177.0854,B 24.9048,C -2.253,E1 24.8415,E2 261.6788} C_DIS
LIN {X -76.7567,Y -12.8451,Z 79,A -175.1228,B 24.9041,C -2.2606,E1 24.8424,E2 259.6862} C_DIS
LIN {X -76.0793,Y -16.3878,Z 79,A -172.6106,B 24.9051,C -2.2489,E1 24.8437,E2 257.1872} C_DIS
LIN {X -75.3347,Y -19.5267,Z 79,A -170.5246,B 24.9063,C -2.2345,E1 24.8451,E2 255.1233} C_DIS
LIN {X -74.3021,Y -23.1472,Z 79,A -167.5784,B 24.9067,C -2.2306,E1 24.8474,E2 252.1696} C_DIS
LIN {X -73.499,Y -25.5835,Z 79,A -165.5845,B 24.9069,C -2.2276,E1 24.8492,E2 250.1714} C_DIS
LIN {X -72.625,Y -27.971,Z 79,A -163.4686,B 24.9069,C -2.2283,E1 24.8513,E2 248.0419} C_DIS
LIN {X -71.2581,Y -31.2875,Z 79,A -160.9684,B 24.9078,C -2.2173,E1 24.854,E2 245.5542} C_DIS
LIN {X -69.951,Y -34.1122,Z 79,A -158.729,B 24.9084,C -2.2096,E1 24.8567,E2 243.3209} C_DIS
LIN {X -68.8275,Y -36.323,Z 79,A -156.3289,B 24.9076,C -2.2192,E1 24.8599,E2 240.8851} C_DIS
LIN {X -65.7634,Y -41.6166,Z 79,A -152.5331,B 24.9101,C -2.1894,E1 24.8652,E2 237.1408} C_DIS
LIN {X -63.8965,Y -44.4276,Z 79,A -149.7546,B 24.91,C -2.1907,E1 24.8696,E2 234.3455} C_DIS
LIN {X -61.9666,Y -47.084,Z 79,A -147.3025,B 24.9104,C -2.1857,E1 24.8737,E2 231.8934} C_DIS
LIN {X -59.8839,Y -49.7041,Z 79,A -145.0391,B 24.9113,C -2.1748,E1 24.8777,E2 229.6455} C_DIS
LIN {X -57.5225,Y -52.4196,Z 79,A -142.2142,B 24.9113,C -2.1734,E1 24.8829,E2 226.8113} C_DIS
LIN {X -54.8722,Y -55.1878,Z 79,A -139.3967,B 24.9119,C -2.1674,E1 24.8884,E2 223.9962} C_DIS
LIN {X -52.4775,Y -57.4694,Z 79,A -136.9866,B 24.9123,C -2.1618,E1 24.8933,E2 221.5894} C_DIS
LIN {X -50.2725,Y -59.4081,Z 79,A -134.9786,B 24.913,C -2.1537,E1 24.8975,E2 219.593} C_DIS
LIN {X -47.0385,Y -62.0008,Z 79,A -131.6712,B 24.913,C -2.1549,E1 24.9048,E2 216.2704} C_DIS
LIN {X -44.3861,Y -63.9254,Z 79,A -129.0549,B 24.9128,C -2.1563,E1 24.9108,E2 213.6417} C_DIS
LIN {X -41.05,Y -66.1175,Z 79,A -126.3018,B 24.9136,C -2.1469,E1 24.9173,E2 210.9022} C_DIS
LIN {X -38.2122,Y -67.7975,Z 79,A -123.8895,B 24.9139,C -2.1431,E1 24.9231,E2 208.4918} C_DIS
LIN {X -35.3167,Y -69.3493,Z 79,A -121.4526,B 24.9141,C -2.1405,E1 24.9291,E2 206.0544} C_DIS
LIN {X -33.0893,Y -70.4397,Z 79,A -119.6532,B 24.9143,C -2.1377,E1 24.9337,E2 204.2571} C_DIS
LIN {X -29.6764,Y -71.9446,Z 79,A -116.9009,B 24.9145,C -2.135,E1 24.9407,E2 201.5048} C_DIS
LIN {X -26.9448,Y -73.0113,Z 79,A -114.739,B 24.9147,C -2.1331,E1 24.9464,E2 199.3429} C_DIS
LIN {X -23.9747,Y -74.0391,Z 79,A -112.4361,B 24.9148,C -2.131,E1 24.9525,E2 197.0408} C_DIS
LIN {X -20.9499,Y -74.9517,Z 79,A -110.0635,B 24.9148,C -2.1307,E1 24.9588,E2 194.665} C_DIS
LIN {X -17.987,Y -75.718,Z 79,A -107.771,B 24.9148,C -2.1305,E1 24.9651,E2 192.3696} C_DIS
LIN {X -14.7311,Y -76.4171,Z 79,A -105.3627,B 24.915,C -2.1284,E1 24.9716,E2 189.9637} C_DIS
LIN {X -11.4831,Y -76.9733,Z 79,A -102.8437,B 24.9149,C -2.1303,E1 24.9786,E2 187.4378} C_DIS
LIN {X -8.1379,Y -77.3974,Z 79,A -100.4449,B 24.9151,C -2.1276,E1 24.9852,E2 185.0439} C_DIS
LIN {X -5.1454,Y -77.6538,Z 79,A -98.2289,B 24.9151,C -2.1277,E1 24.9914,E2 182.8268} C_DIS
LIN {X -2.369,Y -77.788,Z 79,A -96.0934,B 24.9149,C -2.1305,E1 24.9974,E2 180.6843} C_DIS
LIN {X 0.5184,Y -77.8166,Z 79,A -94.6562,B 24.9164,C -2.1115,E1 25.0013,E2 179.2921} C_DIS
Enddeposition()
LIN {X 0.5184,Y -77.8166,Z 79,A -94.6562,B 24.9164,C -2.1115,E1 25.0013,E2 179.2921} C_DIS
Startdeposition()
$VEL.CP = VEL_PRINT
LIN {X -0.6594,Y -76.9096,Z 79,A -96.0758,B 24.9164,C -2.112,E1 24.9973,E2 180.7104} C_DIS
LIN {X -3.5583,Y -76.8302,Z 79,A -98.1627,B 24.9162,C -2.1138,E1 24.9915,E2 182.7934} C_DIS
LIN {X -6.561,Y -76.633,Z 79,A -100.5856,B 24.9166,C -2.1089,E1 24.9847,E2 185.2291} C_DIS
LIN {X -10.3251,Y -76.2173,Z 79,A -103.3925,B 24.9166,C -2.1097,E1 24.9769,E2 188.0359} C_DIS
LIN {X -13.4274,Y -75.7313,Z 79,A -105.569,B 24.9161,C -2.1148,E1 24.971,E2 190.2024} C_DIS
LIN {X -16.404,Y -75.1425,Z 79,A -107.9644,B 24.9163,C -2.1122,E1 24.9644,E2 192.6069} C_DIS
LIN {X -19.7114,Y -74.3443,Z 79,A -110.146,B 24.9155,C -2.123,E1 24.9586,E2 194.7659} C_DIS
LIN {X -21.849,Y -73.7435,Z 79,A -112.0165,B 24.9158,C -2.1183,E1 24.9535,E2 196.6505} C_DIS
LIN {X -24.8025,Y -72.8037,Z 79,A -114.5832,B 24.9162,C -2.1133,E1 24.9466,E2 199.2339} C_DIS
LIN {X -27.8376,Y -71.6983,Z 79,A -117.2791,B 24.9167,C -2.1079,E1 24.9396,E2 201.9482} C_DIS
LIN {X -31.2267,Y -70.289,Z 79,A -119.9509,B 24.9163,C -2.1124,E1 24.9328,E2 204.6156} C_DIS
LIN {X -34.9983,Y -68.488,Z 79,A -122.6884,B 24.9152,C -2.1259,E1 24.926,E2 207.3282} C_DIS
LIN {X -37.8432,Y -66.9592,Z 79,A -125.1181,B 24.915,C -2.1285,E1 24.92,E2 209.7587} C_DIS
LIN {X -40.5601,Y -65.3484,Z 79,A -127.454,B 24.9147,C -2.1324,E1 24.9144,E2 212.0926} C_DIS
LIN {X -44.2785,Y -62.8897,Z 79,A -130.5681,B 24.9139,C -2.1429,E1 24.9073,E2 215.192} C_DIS
LIN {X -47.0038,Y -60.878,Z 79,A -133.8161,B 24.915,C -2.129,E1 24.8999,E2 218.485} C_DIS
LIN {X -50.8388,Y -57.7149,Z 79,A -137.1204,B 24.9136,C -2.146,E1 24.893,E2 221.7615} C_DIS
LIN {X -53.3143,Y -55.4353,Z 79,A -140.1832,B 24.9143,C -2.1372,E1 24.8867,E2 224.8579} C_DIS
LIN {X -55.7045,Y -53.0351,Z 79,A -142.1894,B 24.9129,C -2.1554,E1 24.8829,E2 226.8294} C_DIS
LIN {X -59.2043,Y -49.0951,Z 79,A -145.4794,B 24.9109,C -2.1801,E1 24.8769,E2 230.0752} C_DIS
LIN {X -60.4129,Y -47.6002,Z 79,A -147.4779,B 24.9117,C -2.1693,E1 24.8733,E2 232.1088} C_DIS
LIN {X -62.2804,Y -45.1306,Z 79,A -149.925,B 24.9116,C -2.1715,E1 24.8693,E2 234.5627} C_DIS
LIN {X -64.8081,Y -41.4175,Z 79,A -153.3619,B 24.911,C -2.1777,E1 24.864,E2 238.0018} C_DIS
LIN {X -66.7947,Y -38.1312,Z 79,A -156.0754,B 24.9101,C -2.1888,E1 24.8601,E2 240.7029} C_DIS
LIN {X -68.7228,Y -34.5374,Z 79,A -159.129,B 24.9095,C -2.1967,E1 24.8562,E2 243.754} C_DIS
LIN {X -70.047,Y -31.7637,Z 79,A -161.3493,B 24.9088,C -2.2048,E1 24.8536,E2 245.9671} C_DIS
LIN {X -71.4878,Y -28.3734,Z 79,A -164.0989,B 24.9082,C -2.2124,E1 24.8506,E2 248.7136} C_DIS
LIN {X -72.5192,Y -25.6218,Z 79,A -166.3718,B 24.9078,C -2.2168,E1 24.8485,E2 250.989} C_DIS
LIN {X -74.0353,Y -20.8391,Z 79,A -170.1505,B 24.907,C -2.2269,E1 24.8454,E2 254.7653} C_DIS
LIN {X -74.7203,Y -18.2306,Z 79,A -172.1821,B 24.9065,C -2.2325,E1 24.844,E2 256.7955} C_DIS
LIN {X -75.7753,Y -13.1823,Z 79,A -176.4023,B 24.9063,C -2.2353,E1 24.8417,E2 261.034} C_DIS
LIN {X -76.3718,Y -9.1021,Z 79,A -179.1429,B 24.9048,C -2.2527,E1 24.8407,E2 263.7492} C_DIS
LIN {X -76.6811,Y -5.9595,Z 79,A 178.1669,B 24.9048,C -2.2521,E1 24.8401,E2 266.457} C_DIS
LIN {X -76.9094,Y -0.6909,Z 79,A 174.5841,B 24.9031,C -2.2728,E1 24.8398,E2 270.012} C_DIS
LIN {X -76.8725,Y 2.4731,Z 79,A 171.4903,B 24.9039,C -2.2629,E1 24.84,E2 273.1481} C_DIS
LIN {X -76.6797,Y 5.9771,Z 79,A 169.7009,B 24.9016,C -2.2907,E1 24.8404,E2 274.8819} C_DIS
LIN {X -76.2153,Y 10.3399,Z 79,A 166.4674,B 24.9006,C -2.3019,E1 24.8414,E2 278.108} C_DIS
LIN {X -75.8465,Y 12.7594,Z 79,A 164.4262,B 24.9006,C -2.3025,E1 24.8423,E2 280.1599} C_DIS
LIN {X -75.2459,Y 15.9284,Z 79,A 161.9378,B 24.9001,C -2.308,E1 24.8436,E2 282.6498} C_DIS
LIN {X -73.8895,Y 21.3536,Z 79,A 157.3221,B 24.8998,C -2.3104,E1 24.847,E2 287.2867} C_DIS
LIN {X -72.2705,Y 26.3147,Z 79,A 153.6523,B 24.8984,C -2.3275,E1 24.8503,E2 290.9365} C_DIS
LIN {X -70.9159,Y 29.7729,Z 79,A 151.1426,B 24.8971,C -2.342,E1 24.8529,E2 293.4256} C_DIS
LIN {X -69.6904,Y 32.5383,Z 79,A 148.4038,B 24.8975,C -2.3371,E1 24.8561,E2 296.191} C_DIS
LIN {X -68.2978,Y 35.3705,Z 79,A 146.4294,B 24.8961,C -2.3529,E1 24.8586,E2 298.1383} C_DIS
LIN {X -66.4115,Y 38.7935,Z 79,A 143.2615,B 24.8959,C -2.3551,E1 24.863,E2 301.3174} C_DIS
LIN {X -64.5643,Y 41.7966,Z 79,A 139.9492,B 24.8967,C -2.3461,E1 24.868,E2 304.668} C_DIS
LIN {X -62.1686,Y 45.2833,Z 79,A 136.5279,B 24.8965,C -2.3482,E1 24.8737,E2 308.1009} C_DIS
LIN {X -59.1398,Y 49.1728,Z 79,A 134.1343,B 24.893,C -2.3883,E1 24.8778,E2 310.4098} C_DIS
LIN {X -57.1832,Y 51.4354,Z 79,A 131.6151,B 24.893,C -2.3869,E1 24.8824,E2 312.9439} C_DIS
LIN {X -54.4489,Y 54.3221,Z 79,A 128.1157,B 24.8936,C -2.381,E1 24.8893,E2 316.4722} C_DIS
LIN {X -51.9275,Y 56.7364,Z 79,A 126.4623,B 24.891,C -2.4101,E1 24.8926,E2 318.063} C_DIS
LIN {X -50.1922,Y 58.2786,Z 79,A 124.4261,B 24.8913,C -2.4064,E1 24.8969,E2 320.116} C_DIS
LIN {X -47.5769,Y 60.4313,Z 79,A 122.0673,B 24.8905,C -2.4159,E1 24.902,E2 322.461} C_DIS
LIN {X -44.4665,Y 62.7551,Z 79,A 119.0105,B 24.8903,C -2.4177,E1 24.9089,E2 325.5243} C_DIS
LIN {X -42.2914,Y 64.2411,Z 79,A 116.794,B 24.8905,C -2.4152,E1 24.9141,E2 327.7541} C_DIS
LIN {X -38.6899,Y 66.4737,Z 79,A 113.4658,B 24.8905,C -2.4166,E1 24.9221,E2 331.0892} C_DIS
LIN {X -36.0467,Y 67.9424,Z 79,A 111.2522,B 24.89,C -2.4213,E1 24.9275,E2 333.2978} C_DIS
LIN {X -32.7245,Y 69.6037,Z 79,A 108.7789,B 24.8889,C -2.433,E1 24.9337,E2 335.7495} C_DIS
LIN {X -29.5758,Y 70.999,Z 79,A 106.3512,B 24.8882,C -2.4402,E1 24.9399,E2 338.1659} C_DIS
LIN {X -25.8152,Y 72.4513,Z 79,A 102.7897,B 24.8892,C -2.4298,E1 24.9493,E2 341.7593} C_DIS
LIN {X -18.9692,Y 74.5365,Z 79,A 98.0945,B 24.8872,C -2.4519,E1 24.9617,E2 346.4096} C_DIS
LIN {X -16.8424,Y 75.0466,Z 79,A 96.0422,B 24.888,C -2.4424,E1 24.9674,E2 348.4872} C_DIS
LIN {X -14.1356,Y 75.6032,Z 79,A 94.1441,B 24.8875,C -2.4482,E1 24.9726,E2 350.3737} C_DIS
LIN {X -11.0078,Y 76.1206,Z 79,A 91.874,B 24.8871,C -2.4522,E1 24.9788,E2 352.6361} C_DIS
LIN {X -7.0303,Y 76.5902,Z 79,A 89.2123,B 24.8862,C -2.4624,E1 24.9861,E2 355.2754} C_DIS
LIN {X -3.9985,Y 76.8086,Z 79,A 86.6511,B 24.8868,C -2.4554,E1 24.9933,E2 357.8541} C_DIS
LIN {X -1.1621,Y 76.9038,Z 79,A 84.4935,B 24.8869,C -2.4548,E1 24.9993,E2 360.0133} C_DIS
LIN {X 1.9408,Y 76.8887,Z 79,A 82.1452,B 24.8869,C -2.4541,E1 25.0059,E2 362.3629} C_DIS
LIN {X 5.349,Y 76.7261,Z 79,A 79.5123,B 24.8872,C -2.4517,E1 25.0133,E2 365.0005} C_DIS
LIN {X 8.878,Y 76.3981,Z 79,A 77.013,B 24.8869,C -2.4552,E1 25.0202,E2 367.4899} C_DIS
LIN {X 11.9768,Y 75.9743,Z 79,A 74.6603,B 24.8869,C -2.4539,E1 25.0267,E2 369.8435} C_DIS
LIN {X 15.1479,Y 75.4064,Z 79,A 72.2099,B 24.8872,C -2.4516,E1 25.0334,E2 372.2966} C_DIS
LIN {X 18.5965,Y 74.6311,Z 79,A 69.5837,B 24.8873,C -2.4504,E1 25.0405,E2 374.922} C_DIS
LIN {X 21.522,Y 73.8405,Z 79,A 67.0509,B 24.8882,C -2.4412,E1 25.0474,E2 377.4723} C_DIS
LIN {X 25.1618,Y 72.6806,Z 79,A 63.9662,B 24.889,C -2.4323,E1 25.0556,E2 380.5722} C_DIS
LIN {X 30.196,Y 70.7376,Z 79,A 60.6633,B 24.8875,C -2.4483,E1 25.064,E2 383.8297} C_DIS
LIN {X 32.5244,Y 69.6968,Z 79,A 58.5829,B 24.8882,C -2.441,E1 25.0693,E2 385.922} C_DIS
LIN {X 35.2728,Y 68.3477,Z 79,A 56.5679,B 24.8877,C -2.4457,E1 25.0743,E2 387.9205} C_DIS
LIN {X 37.5168,Y 67.1414,Z 79,A 54.4004,B 24.8887,C -2.4355,E1 25.0797,E2 390.106} C_DIS
LIN {X 41.2145,Y 64.9385,Z 79,A 51.5229,B 24.8883,C -2.4401,E1 25.0865,E2 392.9635} C_DIS
LIN {X 46.5528,Y 61.2252,Z 79,A 46.7014,B 24.8889,C -2.4327,E1 25.0975,E2 397.7859} C_DIS
LIN {X 49.2289,Y 59.0932,Z 79,A 43.9365,B 24.8899,C -2.4218,E1 25.1036,E2 400.5662} C_DIS
LIN {X 51.6631,Y 56.9791,Z 79,A 41.236,B 24.8912,C -2.4084,E1 25.1092,E2 403.2877} C_DIS
LIN {X 54.2495,Y 54.5211,Z 79,A 38.5148,B 24.8918,C -2.401,E1 25.1147,E2 406.0149} C_DIS
LIN {X 56.5945,Y 52.0822,Z 79,A 36.3362,B 24.8914,C -2.4055,E1 25.1188,E2 408.1733} C_DIS
LIN {X 58.7484,Y 49.6407,Z 79,A 33.9408,B 24.8918,C -2.4009,E1 25.1232,E2 410.5689} C_DIS
LIN {X 60.6943,Y 47.2422,Z 79,A 30.9067,B 24.8943,C -2.3739,E1 25.1285,E2 413.6525} C_DIS
LIN {X 62.8874,Y 44.2818,Z 79,A 28.8222,B 24.8931,C -2.3865,E1 25.1318,E2 415.6971} C_DIS
LIN {X 64.7642,Y 41.4859,Z 79,A 25.6867,B 24.8953,C -2.3616,E1 25.1366,E2 418.8757} C_DIS
LIN {X 66.6601,Y 38.3655,Z 79,A 23.8031,B 24.8938,C -2.3792,E1 25.1392,E2 420.708} C_DIS
LIN {X 67.9015,Y 36.1243,Z 79,A 21.8427,B 24.8944,C -2.3725,E1 25.1418,E2 422.6739} C_DIS
LIN {X 69.3091,Y 33.3427,Z 79,A 19.4645,B 24.8951,C -2.3644,E1 25.1448,E2 425.0585} C_DIS
LIN {X 70.7142,Y 30.2515,Z 79,A 16.6,B 24.8966,C -2.3472,E1 25.148,E2 427.948} C_DIS
LIN {X 72.4547,Y 25.8055,Z 79,A 13.6637,B 24.8959,C -2.3556,E1 25.1509,E2 430.8482} C_DIS
LIN {X 73.6043,Y 22.3182,Z 79,A 10.9593,B 24.8965,C -2.3484,E1 25.1532,E2 433.5543} C_DIS
LIN {X 74.5633,Y 18.8646,Z 79,A 8.0754,B 24.8978,C -2.3339,E1 25.1553,E2 436.4559} C_DIS
LIN {X 75.3513,Y 15.4165,Z 79,A 5.5845,B 24.8981,C -2.3302,E1 25.1568,E2 438.941} C_DIS
LIN {X 75.8535,Y 12.7173,Z 79,A 3.5409,B 24.8987,C -2.3239,E1 25.1578,E2 440.9874} C_DIS
LIN {X 76.2946,Y 9.7286,Z 79,A 1.1685,B 24.8996,C -2.3132,E1 25.1587,E2 443.3712} C_DIS
LIN {X 76.6528,Y 6.3135,Z 79,A -1.2761,B 24.9,C -2.3086,E1 25.1594,E2 445.8122} C_DIS
LIN {X 76.8115,Y 3.9459,Z 79,A -3.0972,B 24.9006,C -2.3014,E1 25.1596,E2 447.6395} C_DIS
LIN {X 76.9053,Y 1.0835,Z 79,A -5.2498,B 24.9013,C -2.294,E1 25.1598,E2 449.7968} C_DIS
LIN {X 76.8829,Y -2.1332,Z 79,A -7.8145,B 24.9024,C -2.2812,E1 25.1596,E2 452.3763} C_DIS
LIN {X 76.6701,Y -6.097,Z 79,A -10.5504,B 24.9026,C -2.2786,E1 25.1591,E2 455.1023} C_DIS
LIN {X 76.2433,Y -10.1245,Z 79,A -13.6899,B 24.9037,C -2.2652,E1 25.1581,E2 458.2547} C_DIS
LIN {X 75.8218,Y -12.9068,Z 79,A -15.5458,B 24.9037,C -2.2659,E1 25.1573,E2 460.0981} C_DIS
LIN {X 75.2281,Y -16.0113,Z 79,A -18.283,B 24.9053,C -2.2468,E1 25.1557,E2 462.8644} C_DIS
LIN {X 74.2614,Y -20.0183,Z 79,A -21.0092,B 24.9053,C -2.2476,E1 25.1539,E2 465.573} C_DIS
LIN {X 73.3593,Y -23.1086,Z 79,A -24.1478,B 24.9077,C -2.2178,E1 25.1512,E2 468.7642} C_DIS
LIN {X 72.1336,Y -26.6898,Z 79,A -25.9458,B 24.9059,C -2.2401,E1 25.1496,E2 470.4995} C_DIS
LIN {X 71.1729,Y -29.1535,Z 79,A -28.7811,B 24.9086,C -2.2079,E1 25.1466,E2 473.3951} C_DIS
LIN {X 69.8038,Y -32.2946,Z 79,A -30.5005,B 24.9071,C -2.2254,E1 25.1446,E2 475.0638} C_DIS
LIN {X 68.3857,Y -35.1984,Z 79,A -33.1632,B 24.9083,C -2.2106,E1 25.1413,E2 477.7473} C_DIS
LIN {X 66.9236,Y -37.9053,Z 79,A -35.9623,B 24.9101,C -2.1887,E1 25.1374,E2 480.5835} C_DIS
LIN {X 65.2202,Y -40.7653,Z 79,A -37.3197,B 24.9079,C -2.2156,E1 25.1355,E2 481.8705} C_DIS
LIN {X 64.1197,Y -42.4756,Z 79,A -39.2545,B 24.9093,C -2.1986,E1 25.1325,E2 483.8358} C_DIS
LIN {X 62.3212,Y -45.0749,Z 79,A -42.0318,B 24.9109,C -2.1795,E1 25.128,E2 486.6448} C_DIS
LIN {X 59.5927,Y -48.6236,Z 79,A -44.6803,B 24.9099,C -2.1913,E1 25.1235,E2 489.253} C_DIS
LIN {X 58.1886,Y -50.2963,Z 79,A -46.5989,B 24.911,C -2.1783,E1 25.12,E2 491.1934} C_DIS
LIN {X 56.1964,Y -52.512,Z 79,A -48.7754,B 24.9113,C -2.1741,E1 25.1159,E2 493.3703} C_DIS
LIN {X 53.6939,Y -55.0694,Z 79,A -51.5197,B 24.9121,C -2.1653,E1 25.1104,E2 496.1238} C_DIS
LIN {X 51.8327,Y -56.8235,Z 79,A -53.3401,B 24.9122,C -2.1634,E1 25.1067,E2 497.9412} C_DIS
LIN {X 49.5126,Y -58.8574,Z 79,A -55.6959,B 24.9128,C -2.1565,E1 25.1017,E2 500.3041} C_DIS
LIN {X 46.8433,Y -61.0017,Z 79,A -58.2882,B 24.9133,C -2.1498,E1 25.096,E2 502.9026} C_DIS
LIN {X 43.3952,Y -63.5016,Z 79,A -61.0577,B 24.9129,C -2.1553,E1 25.0897,E2 505.6496} C_DIS
LIN {X 41.4536,Y -64.785,Z 79,A -63.0935,B 24.9139,C -2.1431,E1 25.0849,E2 507.7076} C_DIS
LIN {X 38.7345,Y -66.4479,Z 79,A -65.4784,B 24.9142,C -2.1384,E1 25.0792,E2 510.0962} C_DIS
LIN {X 35.7138,Y -68.1177,Z 79,A -67.9965,B 24.9145,C -2.1356,E1 25.073,E2 512.6138} C_DIS
LIN {X 32.6571,Y -69.6351,Z 79,A -70.2463,B 24.9141,C -2.14,E1 25.0674,E2 514.8471} C_DIS
LIN {X 29.3797,Y -71.0806,Z 79,A -73.8278,B 24.9165,C -2.1098,E1 25.058,E2 518.4916} C_DIS
LIN {X 26.1865,Y -72.3172,Z 79,A -75.4761,B 24.9147,C -2.1323,E1 25.0539,E2 520.0832} C_DIS
LIN {X 21.4801,Y -73.8529,Z 79,A -79.1752,B 24.9151,C -2.1276,E1 25.044,E2 523.7866} C_DIS
LIN {X 19.1473,Y -74.4907,Z 79,A -81.1399,B 24.9156,C -2.121,E1 25.0387,E2 525.7637} C_DIS
LIN {X 16.1144,Y -75.2056,Z 79,A -83.9041,B 24.9168,C -2.1064,E1 25.0311,E2 528.5589} C_DIS
LIN {X 11.7561,Y -76.0084,Z 79,A -86.7934,B 24.9161,C -2.1155,E1 25.0232,E2 531.4237} C_DIS
LIN {X 8.7732,Y -76.4104,Z 79,A -89.0944,B 24.9163,C -2.1124,E1 25.0168,E2 533.7302} C_DIS
LIN {X 5.4758,Y -76.7175,Z 79,A -91.6685,B 24.9166,C -2.1083,E1 25.0096,E2 536.3128} C_DIS
LIN {X 1.651,Y -76.8948,Z 79,A -94.0168,B 24.9156,C -2.1212,E1 25.0031,E2 538.6297} C_DIS
LIN {X 1.651,Y -76.8948,Z 79,A -94.0168,B 24.9156,C -2.1212,E1 25.0031,E2 538.6297} C_DIS
Enddeposition()
LIN {X 0.517,Y -75.9957,Z 79,A -95.0147,B 24.9147,C -2.1328,E1 25.0004,E2 539.6} C_DIS
Startdeposition()
$VEL.CP = VEL_PRINT
LIN {X 3.6805,Y -75.9123,Z 79,A -91.3572,B 24.9118,C -2.1688,E1 25.0109,E2 535.858} C_DIS
LIN {X 7.7311,Y -75.6063,Z 79,A -88.7582,B 24.9127,C -2.1573,E1 25.018,E2 533.2876} C_DIS
LIN {X 10.6071,Y -75.2565,Z 79,A -86.6573,B 24.9127,C -2.1564,E1 25.0238,E2 531.1907} C_DIS
LIN {X 13.9684,Y -74.7067,Z 79,A -83.7076,B 24.9117,C -2.1692,E1 25.032,E2 528.2138} C_DIS
LIN {X 18.4385,Y -73.731,Z 79,A -80.4598,B 24.9119,C -2.1667,E1 25.0408,E2 524.9765} C_DIS
LIN {X 20.7883,Y -73.102,Z 79,A -78.3487,B 24.9111,C -2.1767,E1 25.0465,E2 522.8452} C_DIS
LIN {X 25.3991,Y -71.6309,Z 79,A -75.2511,B 24.9121,C -2.1652,E1 25.0547,E2 519.7807} C_DIS
LIN {X 28.8963,Y -70.2931,Z 79,A -71.8531,B 24.9104,C -2.1858,E1 25.0636,E2 516.3416} C_DIS
LIN {X 32.0604,Y -68.907,Z 79,A -69.848,B 24.9115,C -2.1723,E1 25.0686,E2 514.3734} C_DIS
LIN {X 36.2038,Y -66.8231,Z 79,A -65.9008,B 24.9099,C -2.1913,E1 25.0785,E2 510.3922} C_DIS
LIN {X 39.5132,Y -64.9211,Z 79,A -63.2198,B 24.9099,C -2.1907,E1 25.0849,E2 507.7208} C_DIS
LIN {X 41.9985,Y -63.342,Z 79,A -60.3679,B 24.9081,C -2.2138,E1 25.0916,E2 504.8237} C_DIS
LIN {X 44.8845,Y -61.3304,Z 79,A -58.0105,B 24.9083,C -2.2104,E1 25.0969,E2 502.4826} C_DIS
LIN {X 48.3161,Y -58.6661,Z 79,A -55.1373,B 24.9088,C -2.2055,E1 25.1031,E2 499.6319} C_DIS
LIN {X 50.8121,Y -56.5172,Z 79,A -53.0247,B 24.9092,C -2.2001,E1 25.1075,E2 497.5404} C_DIS
LIN {X 53.1799,Y -54.2959,Z 79,A -49.8035,B 24.9068,C -2.2291,E1 25.1141,E2 494.264} C_DIS
LIN {X 56.19,Y -51.1743,Z 79,A -47.026,B 24.9074,C -2.2223,E1 25.1194,E2 491.5146} C_DIS
LIN {X 58.2182,Y -48.8551,Z 79,A -44.985,B 24.9076,C -2.2198,E1 25.1231,E2 489.4888} C_DIS
LIN {X 60.273,Y -46.295,Z 79,A -42.0596,B 24.9059,C -2.2399,E1 25.1282,E2 486.5296} C_DIS
LIN {X 62.7818,Y -42.8318,Z 79,A -39.0198,B 24.9056,C -2.2431,E1 25.1331,E2 483.4971} C_DIS
LIN {X 64.2142,Y -40.6546,Z 79,A -36.2689,B 24.9031,C -2.2727,E1 25.1373,E2 480.6903} C_DIS
LIN {X 66.1706,Y -37.3836,Z 79,A -34.4942,B 24.9053,C -2.2473,E1 25.1396,E2 478.9846} C_DIS
LIN {X 68.2313,Y -33.4748,Z 79,A -31.1409,B 24.9044,C -2.2577,E1 25.144,E2 475.6245} C_DIS
LIN {X 69.0801,Y -31.6883,Z 79,A -29.1167,B 24.9026,C -2.2784,E1 25.1464,E2 473.5623} C_DIS
LIN {X 71.0474,Y -26.9872,Z 79,A -25.4287,B 24.902,C -2.2854,E1 25.1502,E2 469.8783} C_DIS
LIN {X 72.8221,Y -21.7485,Z 79,A -21.519,B 24.9016,C -2.2902,E1 25.1536,E2 465.9793} C_DIS
LIN {X 73.3868,Y -19.7592,Z 79,A -19.1292,B 24.8989,C -2.3208,E1 25.1553,E2 463.5311} C_DIS
LIN {X 74.2873,Y -16.046,Z 79,A -16.7952,B 24.8996,C -2.3129,E1 25.1567,E2 461.2292} C_DIS
LIN {X 75.0368,Y -12.0724,Z 79,A -13.9558,B 24.8994,C -2.3161,E1 25.1581,E2 458.3989} C_DIS
LIN {X 75.5302,Y -8.4488,Z 79,A -11.3244,B 24.8989,C -2.321,E1 25.159,E2 455.7714} C_DIS
LIN {X 75.8655,Y -4.5383,Z 79,A -7.9839,B 24.8971,C -2.3422,E1 25.1596,E2 452.4007} C_DIS
LIN {X 75.9999,Y -0.2966,Z 79,A -5.1722,B 24.8972,C -2.3405,E1 25.1598,E2 449.6099} C_DIS
LIN {X 75.9471,Y 2.8698,Z 79,A -2.9437,B 24.897,C -2.3432,E1 25.1596,E2 447.3882} C_DIS
LIN {X 75.7557,Y 6.0926,Z 79,A -0.1237,B 24.8952,C -2.3627,E1 25.1591,E2 444.5388} C_DIS
LIN {X 75.342,Y 9.9836,Z 79,A 2.4944,B 24.8953,C -2.3618,E1 25.1582,E2 441.9384} C_DIS
LIN {X 74.8714,Y 13.0571,Z 79,A 5.1312,B 24.8939,C -2.378,E1 25.157,E2 439.2787} C_DIS
LIN {X 73.9333,Y 17.6092,Z 79,A 8.4149,B 24.8935,C -2.382,E1 25.155,E2 436.0048} C_DIS
LIN {X 73.1355,Y 20.6699,Z 79,A 10.5012,B 24.8937,C -2.3801,E1 25.1535,E2 433.9348} C_DIS
LIN {X 71.6147,Y 25.4453,Z 79,A 14.064,B 24.8933,C -2.3847,E1 25.1505,E2 430.3814} C_DIS
LIN {X 70.1245,Y 29.3027,Z 79,A 17.5272,B 24.8915,C -2.4041,E1 25.1469,E2 426.8915} C_DIS
LIN {X 68.7068,Y 32.4901,Z 79,A 20.175,B 24.8908,C -2.412,E1 25.1438,E2 424.2394} C_DIS
LIN {X 67.4028,Y 35.1145,Z 79,A 22.3752,B 24.8903,C -2.4178,E1 25.141,E2 422.0373} C_DIS
LIN {X 65.6414,Y 38.306,Z 79,A 25.428,B 24.8888,C -2.4343,E1 25.1367,E2 418.9613} C_DIS
LIN {X 62.6887,Y 42.9693,Z 79,A 29.6107,B 24.8878,C -2.4455,E1 25.1303,E2 414.773} C_DIS
LIN {X 59.346,Y 47.4794,Z 79,A 33.5061,B 24.8878,C -2.4455,E1 25.1238,E2 410.8958} C_DIS
LIN {X 57.3707,Y 49.8466,Z 79,A 35.7367,B 24.8875,C -2.4481,E1 25.1197,E2 408.6693} C_DIS
LIN {X 53.5364,Y 53.9438,Z 79,A 39.94,B 24.8867,C -2.4564,E1 25.1116,E2 404.4646} C_DIS
LIN {X 50.5463,Y 56.7553,Z 79,A 43.1089,B 24.886,C -2.4648,E1 25.1051,E2 401.2887} C_DIS
LIN {X 48.0601,Y 58.8756,Z 79,A 45.4797,B 24.8858,C -2.4667,E1 25.1,E2 398.9224} C_DIS
LIN {X 46.3762,Y 60.2104,Z 79,A 47.564,B 24.8843,C -2.4832,E1 25.0953,E2 396.8069} C_DIS
LIN {X 41.8096,Y 63.4666,Z 79,A 51.0702,B 24.8856,C -2.4692,E1 25.0874,E2 393.3458} C_DIS
LIN {X 38.2658,Y 65.6657,Z 79,A 54.5586,B 24.8842,C -2.4837,E1 25.079,E2 389.834} C_DIS
LIN {X 35.4254,Y 67.239,Z 79,A 56.6905,B 24.8847,C -2.478,E1 25.0738,E2 387.7217} C_DIS
LIN {X 33.6042,Y 68.1677,Z 79,A 58.4587,B 24.884,C -2.4863,E1 25.0694,E2 385.9385} C_DIS
LIN {X 30.5069,Y 69.6089,Z 79,A 61.6551,B 24.882,C -2.5069,E1 25.0611,E2 382.7013} C_DIS
LIN {X 27.3623,Y 70.9053,Z 79,A 64.2834,B 24.8816,C -2.5111,E1 25.0543,E2 380.0687} C_DIS
LIN {X 24.0707,Y 72.0881,Z 79,A 66.003,B 24.8839,C -2.4876,E1 25.0499,E2 378.4083} C_DIS
LIN {X 20.3734,Y 73.2195,Z 79,A 69.1473,B 24.8831,C -2.496,E1 25.0414,E2 375.2495} C_DIS
LIN {X 17.3646,Y 73.9905,Z 79,A 71.9286,B 24.8818,C -2.5095,E1 25.0338,E2 372.44} C_DIS
LIN {X 12.1854,Y 75.0179,Z 79,A 75.4737,B 24.8828,C -2.499,E1 25.0241,E2 368.9239} C_DIS
LIN {X 9.0592,Y 75.4588,Z 79,A 77.752,B 24.883,C -2.4967,E1 25.0178,E2 366.6529} C_DIS
LIN {X 4.8294,Y 75.8473,Z 79,A 81.412,B 24.8818,C -2.5093,E1 25.0076,E2 362.9647} C_DIS
LIN {X 0.5044,Y 75.9986,Z 79,A 84.2795,B 24.8828,C -2.4982,E1 24.9996,E2 360.124} C_DIS
LIN {X -2.5663,Y 75.9573,Z 79,A 86.3317,B 24.8836,C -2.4906,E1 24.994,E2 358.0899} C_DIS
LIN {X -6.6953,Y 75.7054,Z 79,A 89.3792,B 24.8839,C -2.4874,E1 24.9855,E2 355.0489} C_DIS
LIN {X -10.2352,Y 75.3093,Z 79,A 92.4817,B 24.883,C -2.4969,E1 24.9768,E2 351.9218} C_DIS
LIN {X -13.5458,Y 74.7835,Z 79,A 94.7196,B 24.8839,C -2.4875,E1 24.9707,E2 349.7041} C_DIS
LIN {X -17.5987,Y 73.9349,Z 79,A 97.9027,B 24.8839,C -2.4864,E1 24.962,E2 346.5197} C_DIS
LIN {X -20.8139,Y 73.0947,Z 79,A 100.8727,B 24.8831,C -2.4959,E1 24.954,E2 343.5224} C_DIS
LIN {X -24.5693,Y 71.92,Z 79,A 104.2225,B 24.8825,C -2.5023,E1 24.945,E2 340.151} C_DIS
LIN {X -27.7594,Y 70.7493,Z 79,A 106.3408,B 24.8839,C -2.4875,E1 24.9396,E2 338.0636} C_DIS
LIN {X -31.2989,Y 69.2563,Z 79,A 109.0592,B 24.8847,C -2.4787,E1 24.9327,E2 335.3597} C_DIS
LIN {X -36.3743,Y 66.7307,Z 79,A 113.398,B 24.8852,C -2.4734,E1 24.9219,E2 331.0218} C_DIS
LIN {X -40.0808,Y 64.5726,Z 79,A 116.9922,B 24.8849,C -2.4767,E1 24.9133,E2 327.4087} C_DIS
LIN {X -43.4291,Y 62.3696,Z 79,A 119.817,B 24.8859,C -2.4658,E1 24.9068,E2 324.6003} C_DIS
LIN {X -46.6038,Y 60.035,Z 79,A 122.8901,B 24.8862,C -2.4622,E1 24.8999,E2 321.5247} C_DIS
LIN {X -50.7306,Y 56.5902,Z 79,A 127.0672,B 24.8868,C -2.4563,E1 24.8911,E2 317.3454} C_DIS
LIN {X -54.6325,Y 52.8333,Z 79,A 130.952,B 24.8881,C -2.4416,E1 24.8835,E2 313.4792} C_DIS
LIN {X -58.1843,Y 48.8959,Z 79,A 134.5361,B 24.89,C -2.4214,E1 24.8769,E2 309.9272} C_DIS
LIN {X -60.1441,Y 46.4622,Z 79,A 137.3929,B 24.8894,C -2.4275,E1 24.8719,E2 307.0425} C_DIS
LIN {X -62.3688,Y 43.4302,Z 79,A 140.0523,B 24.8905,C -2.4156,E1 24.8676,E2 304.3985} C_DIS
LIN {X -63.9285,Y 41.0999,Z 79,A 141.9689,B 24.8915,C -2.4049,E1 24.8647,E2 302.4977} C_DIS
LIN {X -65.6122,Y 38.3558,Z 79,A 144.9087,B 24.891,C -2.4105,E1 24.8604,E2 299.5295} C_DIS
LIN {X -67.3214,Y 35.269,Z 79,A 148.1827,B 24.8903,C -2.4178,E1 24.8562,E2 296.2207} C_DIS
LIN {X -69.1515,Y 31.5315,Z 79,A 150.4556,B 24.893,C -2.3874,E1 24.8536,E2 294.0078} C_DIS
LIN {X -70.3901,Y 28.658,Z 79,A 153.4446,B 24.8923,C -2.3956,E1 24.8503,E2 290.9827} C_DIS
LIN {X -71.6052,Y 25.4726,Z 79,A 156.3928,B 24.8922,C -2.3969,E1 24.8476,E2 288.0146} C_DIS
LIN {X -72.9562,Y 21.2966,Z 79,A 158.3792,B 24.896,C -2.3547,E1 24.8461,E2 286.1175} C_DIS
LIN {X -73.9978,Y 17.3329,Z 79,A 161.438,B 24.8969,C -2.3443,E1 24.8439,E2 283.0658} C_DIS
LIN {X -74.5271,Y 14.8966,Z 79,A 163.7395,B 24.8965,C -2.3484,E1 24.8426,E2 280.7408} C_DIS
LIN {X -75.1241,Y 11.5075,Z 79,A 167.5116,B 24.8947,C -2.3687,E1 24.8409,E2 276.8978} C_DIS
LIN {X -75.7084,Y 6.6621,Z 79,A 169.6863,B 24.8989,C -2.3207,E1 24.8404,E2 274.8248} C_DIS
LIN {X -75.9227,Y 3.4382,Z 79,A 172.9107,B 24.898,C -2.3318,E1 24.8398,E2 271.5544} C_DIS
LIN {X -76.0002,Y 0.243,Z 79,A 175.1704,B 24.899,C -2.3206,E1 24.8398,E2 269.3081} C_DIS
LIN {X -75.9008,Y -3.8994,Z 79,A 178.1087,B 24.9002,C -2.3062,E1 24.8401,E2 266.3864} C_DIS
LIN {X -75.6125,Y -7.6712,Z 79,A -179.0649,B 24.901,C -2.2966,E1 24.8408,E2 263.5658} C_DIS
LIN {X -75.0643,Y -11.8856,Z 79,A -175.8251,B 24.9018,C -2.2875,E1 24.842,E2 260.3285} C_DIS
LIN {X -74.388,Y -15.5693,Z 79,A -172.5046,B 24.9015,C -2.2909,E1 24.8439,E2 256.9804} C_DIS
LIN {X -72.9231,Y -21.4081,Z 79,A -168.0746,B 24.9029,C -2.2745,E1 24.8471,E2 252.5636} C_DIS
LIN {X -71.5878,Y -25.5219,Z 79,A -165.3151,B 24.9048,C -2.2528,E1 24.8495,E2 249.8404} C_DIS
LIN {X -70.5692,Y -28.218,Z 79,A -162.4946,B 24.904,C -2.2623,E1 24.8524,E2 246.9813} C_DIS
LIN {X -68.743,Y -32.4128,Z 79,A -159.4407,B 24.9056,C -2.2429,E1 24.8559,E2 243.9569} C_DIS
LIN {X -66.3161,Y -37.1245,Z 79,A -156.0717,B 24.9078,C -2.2168,E1 24.8603,E2 240.6324} C_DIS
LIN {X -64.228,Y -40.6325,Z 79,A -152.5602,B 24.9076,C -2.2193,E1 24.8653,E2 237.0968} C_DIS
LIN {X -62.4044,Y -43.379,Z 79,A -149.6212,B 24.9072,C -2.2243,E1 24.87,E2 234.1313} C_DIS
LIN {X -60.1203,Y -46.4932,Z 79,A -147.1275,B 24.9086,C -2.2069,E1 24.8741,E2 231.667} C_DIS
LIN {X -57.8266,Y -49.3166,Z 79,A -143.7836,B 24.9079,C -2.2157,E1 24.8801,E2 228.2869} C_DIS
LIN {X -55.044,Y -52.4063,Z 79,A -140.674,B 24.9085,C -2.2082,E1 24.8861,E2 225.1816} C_DIS
LIN {X -51.0988,Y -56.2593,Z 79,A -136.8273,B 24.9099,C -2.1919,E1 24.8938,E2 221.3579} C_DIS
LIN {X -49.1482,Y -57.9701,Z 79,A -134.2495,B 24.9089,C -2.2041,E1 24.8994,E2 218.7409} C_DIS
LIN {X -46.5518,Y -60.0747,Z 79,A -131.8984,B 24.9096,C -2.1953,E1 24.9045,E2 216.4022} C_DIS
LIN {X -43.1656,Y -62.5527,Z 79,A -129.3941,B 24.9114,C -2.173,E1 24.9101,E2 213.9423} C_DIS
LIN {X -40.9756,Y -64.0082,Z 79,A -127.1967,B 24.9112,C -2.1755,E1 24.9153,E2 211.7318} C_DIS
LIN {X -38.2335,Y -65.6843,Z 79,A -124.7728,B 24.9115,C -2.1721,E1 24.9211,E2 209.3087} C_DIS
LIN {X -35.6194,Y -67.1368,Z 79,A -122.5084,B 24.9117,C -2.1694,E1 24.9267,E2 207.0444} C_DIS
LIN {X -33.6976,Y -68.1213,Z 79,A -120.1466,B 24.9103,C -2.1868,E1 24.9327,E2 204.635} C_DIS
LIN {X -30.4417,Y -69.6373,Z 79,A -118.4796,B 24.9128,C -2.1563,E1 24.9368,E2 203.0365} C_DIS
LIN {X -27.0411,Y -71.0271,Z 79,A -115.5567,B 24.9127,C -2.1576,E1 24.9444,E2 200.1039} C_DIS
LIN {X -23.642,Y -72.2299,Z 79,A -112.6592,B 24.9125,C -2.1601,E1 24.952,E2 197.1949} C_DIS
LIN {X -20.5909,Y -73.1579,Z 79,A -110.5926,B 24.9133,C -2.1495,E1 24.9575,E2 195.1501} C_DIS
LIN {X -17.5914,Y -73.9375,Z 79,A -107.7492,B 24.9123,C -2.1618,E1 24.9653,E2 192.2735} C_DIS
LIN {X -14.0059,Y -74.6995,Z 79,A -105.0898,B 24.9127,C -2.1579,E1 24.9726,E2 189.6204} C_DIS
LIN {X -10.8118,Y -75.2274,Z 79,A -103.0228,B 24.9135,C -2.1471,E1 24.9782,E2 187.5771} C_DIS
LIN {X -7.9625,Y -75.5821,Z 79,A -100.2196,B 24.9121,C -2.1643,E1 24.9861,E2 184.7313} C_DIS
LIN {X -3.8445,Y -75.9038,Z 79,A -97.3818,B 24.9128,C -2.1567,E1 24.994,E2 181.9105} C_DIS
LIN {X -0.8439,Y -75.9965,Z 79,A -95.0752,B 24.9126,C -2.1583,E1 25.0004,E2 179.6} C_DIS
LIN {X -0.8439,Y -75.9965,Z 79,A -95.0752,B 24.9126,C -2.1583,E1 25.0004,E2 179.6} C_DIS
Enddeposition()
LIN {X 0.4928,Y -75.0785,Z 79,A -93.6629,B 24.9104,C -2.1855,E1 25.0046,E2 178.1233} C_DIS
Startdeposition()
$VEL.CP = VEL_PRINT
LIN {X -1.0287,Y -75.0822,Z 79,A -96.4754,B 24.9141,C -2.1401,E1 24.9964,E2 181.0436} C_DIS
LIN {X -4.1317,Y -74.9747,Z 79,A -98.7274,B 24.9139,C -2.143,E1 24.9901,E2 183.2891} C_DIS
LIN {X -7.5261,Y -74.7109,Z 79,A -101.9406,B 24.9152,C -2.1269,E1 24.9811,E2 186.5422} C_DIS
LIN {X -12.0501,Y -74.116,Z 79,A -104.9172,B 24.914,C -2.1409,E1 24.9729,E2 189.4879} C_DIS
LIN {X -14.4578,Y -73.6839,Z 79,A -107.1771,B 24.9148,C -2.1314,E1 24.9667,E2 191.773} C_DIS
LIN {X -20.394,Y -72.2659,Z 79,A -111.4371,B 24.9138,C -2.1443,E1 24.9552,E2 196.0084} C_DIS
LIN {X -22.4669,Y -71.6489,Z 79,A -113.1133,B 24.9138,C -2.1448,E1 24.9507,E2 197.6863} C_DIS
LIN {X -26.4466,Y -70.2771,Z 79,A -116.3774,B 24.9136,C -2.1462,E1 24.9421,E2 200.9535} C_DIS
LIN {X -29.874,Y -68.89,Z 79,A -120.2737,B 24.9155,C -2.1221,E1 24.932,E2 204.9163} C_DIS
LIN {X -34.1445,Y -66.8762,Z 79,A -122.6453,B 24.9127,C -2.1573,E1 24.9262,E2 207.2104} C_DIS
LIN {X -36.7579,Y -65.4764,Z 79,A -125.0308,B 24.9127,C -2.1572,E1 24.9204,E2 209.6029} C_DIS
LIN {X -40.0468,Y -63.5187,Z 79,A -127.6264,B 24.9117,C -2.1696,E1 24.9142,E2 212.1771} C_DIS
LIN {X -42.3072,Y -62.0358,Z 79,A -129.8999,B 24.9119,C -2.1675,E1 24.9089,E2 214.4629} C_DIS
LIN {X -44.0346,Y -60.8226,Z 79,A -132.1029,B 24.9128,C -2.1556,E1 24.9039,E2 216.702} C_DIS
LIN {X -48.6453,Y -57.2006,Z 79,A -135.8291,B 24.9107,C -2.1821,E1 24.8959,E2 220.3789} C_DIS
LIN {X -51.9853,Y -54.1833,Z 79,A -140.2826,B 24.9122,C -2.1642,E1 24.8866,E2 224.8933} C_DIS
LIN {X -54.4801,Y -51.6748,Z 79,A -142.218,B 24.9102,C -2.1884,E1 24.883,E2 226.7794} C_DIS
LIN {X -57.8764,Y -47.8387,Z 79,A -146.2877,B 24.9098,C -2.1933,E1 24.8755,E2 230.8557} C_DIS
LIN {X -59.497,Y -45.808,Z 79,A -148.6719,B 24.9102,C -2.1884,E1 24.8714,E2 233.263} C_DIS
LIN {X -62.7428,Y -41.2508,Z 79,A -152.5598,B 24.9085,C -2.2081,E1 24.8653,E2 237.1231} C_DIS
LIN {X -65.3102,Y -37.0534,Z 79,A -156.5549,B 24.9082,C -2.2123,E1 24.8596,E2 241.1289} C_DIS
LIN {X -67.5262,Y -32.8423,Z 79,A -159.9101,B 24.9068,C -2.2287,E1 24.8553,E2 244.4629} C_DIS
LIN {X -69.6481,Y -28.0621,Z 79,A -164.3364,B 24.9068,C -2.2298,E1 24.8504,E2 248.9111} C_DIS
LIN {X -71.0624,Y -24.2587,Z 79,A -166.7111,B 24.9045,C -2.2557,E1 24.8482,E2 251.2374} C_DIS
LIN {X -72.5562,Y -19.3373,Z 79,A -171.0418,B 24.9044,C -2.2579,E1 24.8448,E2 255.5878} C_DIS
LIN {X -73.4777,Y -15.468,Z 79,A -174.1159,B 24.9037,C -2.2662,E1 24.8429,E2 258.66} C_DIS
LIN {X -74.1869,Y -11.6008,Z 79,A -177.5256,B 24.9037,C -2.2661,E1 24.8413,E2 262.0904} C_DIS
LIN {X -74.829,Y -6.2348,Z 79,A 178.5894,B 24.9021,C -2.2845,E1 24.8402,E2 265.9547} C_DIS
LIN {X -75.0455,Y -2.5049,Z 79,A 175.5307,B 24.9017,C -2.2888,E1 24.8398,E2 269.0215} C_DIS
LIN {X -75.0795,Y 1.178,Z 79,A 172.5942,B 24.9012,C -2.2948,E1 24.8398,E2 271.9614} C_DIS
LIN {X -74.8057,Y 6.5208,Z 79,A 168.3853,B 24.9003,C -2.3049,E1 24.8407,E2 276.1715} C_DIS
Enddeposition()
END
